    {attribute	'TcLinkTo'	:=	'.Status:=TIIB[K4S8_DRL_03_E18_EL6021]^COM TxPDO-Map Inputs^Status;
                                 .D[0]:=TIIB[K4S8_DRL_03_E18_EL6021]^COM TxPDO-Map Inputs^Data In 0;
                                 .D[1]:=TIIB[K4S8_DRL_03_E18_EL6021]^COM TxPDO-Map Inputs^Data In 1;
                                 .D[2]:=TIIB[K4S8_DRL_03_E18_EL6021]^COM TxPDO-Map Inputs^Data In 2;
                                 .D[3]:=TIIB[K4S8_DRL_03_E18_EL6021]^COM TxPDO-Map Inputs^Data In 3;
                                 .D[4]:=TIIB[K4S8_DRL_03_E18_EL6021]^COM TxPDO-Map Inputs^Data In 4;
                                 .D[5]:=TIIB[K4S8_DRL_03_E18_EL6021]^COM TxPDO-Map Inputs^Data In 5;
                                 .D[6]:=TIIB[K4S8_DRL_03_E18_EL6021]^COM TxPDO-Map Inputs^Data In 6;
                                 .D[7]:=TIIB[K4S8_DRL_03_E18_EL6021]^COM TxPDO-Map Inputs^Data In 7;
                                 .D[8]:=TIIB[K4S8_DRL_03_E18_EL6021]^COM TxPDO-Map Inputs^Data In 8;
                                 .D[9]:=TIIB[K4S8_DRL_03_E18_EL6021]^COM TxPDO-Map Inputs^Data In 9;
                                 .D[10]:=TIIB[K4S8_DRL_03_E18_EL6021]^COM TxPDO-Map Inputs^Data In 10;
                                 .D[11]:=TIIB[K4S8_DRL_03_E18_EL6021]^COM TxPDO-Map Inputs^Data In 11;
                                 .D[12]:=TIIB[K4S8_DRL_03_E18_EL6021]^COM TxPDO-Map Inputs^Data In 12;
                                 .D[13]:=TIIB[K4S8_DRL_03_E18_EL6021]^COM TxPDO-Map Inputs^Data In 13;
                                 .D[14]:=TIIB[K4S8_DRL_03_E18_EL6021]^COM TxPDO-Map Inputs^Data In 14;
                                 .D[15]:=TIIB[K4S8_DRL_03_E18_EL6021]^COM TxPDO-Map Inputs^Data In 15;
                                 .D[16]:=TIIB[K4S8_DRL_03_E18_EL6021]^COM TxPDO-Map Inputs^Data In 16;
                                 .D[17]:=TIIB[K4S8_DRL_03_E18_EL6021]^COM TxPDO-Map Inputs^Data In 17;
                                 .D[18]:=TIIB[K4S8_DRL_03_E18_EL6021]^COM TxPDO-Map Inputs^Data In 18;
                                 .D[19]:=TIIB[K4S8_DRL_03_E18_EL6021]^COM TxPDO-Map Inputs^Data In 19;
                                 .D[20]:=TIIB[K4S8_DRL_03_E18_EL6021]^COM TxPDO-Map Inputs^Data In 20;
                                 .D[21]:=TIIB[K4S8_DRL_03_E18_EL6021]^COM TxPDO-Map Inputs^Data In 21
    '}
    stComIn_DREAM_DP1_PTM_01 AT %I* : EL6inData22B;

    {attribute 'TcLinkTo'	:=	'.Ctrl:=TIIB[K4S8_DRL_03_E18_EL6021]^COM RxPDO-Map Outputs^Ctrl;
                                 .D[0]:=TIIB[K4S8_DRL_03_E18_EL6021]^COM RxPDO-Map Outputs^Data Out 0;
                                 .D[1]:=TIIB[K4S8_DRL_03_E18_EL6021]^COM RxPDO-Map Outputs^Data Out 1;
                                 .D[2]:=TIIB[K4S8_DRL_03_E18_EL6021]^COM RxPDO-Map Outputs^Data Out 2;
                                 .D[3]:=TIIB[K4S8_DRL_03_E18_EL6021]^COM RxPDO-Map Outputs^Data Out 3;
                                 .D[4]:=TIIB[K4S8_DRL_03_E18_EL6021]^COM RxPDO-Map Outputs^Data Out 4;
                                 .D[5]:=TIIB[K4S8_DRL_03_E18_EL6021]^COM RxPDO-Map Outputs^Data Out 5;
                                 .D[6]:=TIIB[K4S8_DRL_03_E18_EL6021]^COM RxPDO-Map Outputs^Data Out 6;
                                 .D[7]:=TIIB[K4S8_DRL_03_E18_EL6021]^COM RxPDO-Map Outputs^Data Out 7;
                                 .D[8]:=TIIB[K4S8_DRL_03_E18_EL6021]^COM RxPDO-Map Outputs^Data Out 8;
                                 .D[9]:=TIIB[K4S8_DRL_03_E18_EL6021]^COM RxPDO-Map Outputs^Data Out 9;
                                 .D[10]:=TIIB[K4S8_DRL_03_E18_EL6021]^COM RxPDO-Map Outputs^Data Out 10;
                                 .D[11]:=TIIB[K4S8_DRL_03_E18_EL6021]^COM RxPDO-Map Outputs^Data Out 11;
                                 .D[12]:=TIIB[K4S8_DRL_03_E18_EL6021]^COM RxPDO-Map Outputs^Data Out 12;
                                 .D[13]:=TIIB[K4S8_DRL_03_E18_EL6021]^COM RxPDO-Map Outputs^Data Out 13;
                                 .D[14]:=TIIB[K4S8_DRL_03_E18_EL6021]^COM RxPDO-Map Outputs^Data Out 14;
                                 .D[15]:=TIIB[K4S8_DRL_03_E18_EL6021]^COM RxPDO-Map Outputs^Data Out 15;
                                 .D[16]:=TIIB[K4S8_DRL_03_E18_EL6021]^COM RxPDO-Map Outputs^Data Out 16;
                                 .D[17]:=TIIB[K4S8_DRL_03_E18_EL6021]^COM RxPDO-Map Outputs^Data Out 17;
                                 .D[18]:=TIIB[K4S8_DRL_03_E18_EL6021]^COM RxPDO-Map Outputs^Data Out 18;
                                 .D[19]:=TIIB[K4S8_DRL_03_E18_EL6021]^COM RxPDO-Map Outputs^Data Out 19;
                                 .D[20]:=TIIB[K4S8_DRL_03_E18_EL6021]^COM RxPDO-Map Outputs^Data Out 20;
                                 .D[21]:=TIIB[K4S8_DRL_03_E18_EL6021]^COM RxPDO-Map Outputs^Data Out 21
    '}
    stComOut_DREAM_DP1_PTM_01 AT %Q* : EL6outData22B;

    {attribute	'TcLinkTo'	:=	'.Status:=TIIB[R20_DRL_03_E9_EL6001]^COM Inputs^Status;
                                 .D[0]:=TIIB[R20_DRL_03_E9_EL6001]^COM Inputs^Data In 0;
                                 .D[1]:=TIIB[R20_DRL_03_E9_EL6001]^COM Inputs^Data In 1;
                                 .D[2]:=TIIB[R20_DRL_03_E9_EL6001]^COM Inputs^Data In 2;
                                 .D[3]:=TIIB[R20_DRL_03_E9_EL6001]^COM Inputs^Data In 3;
                                 .D[4]:=TIIB[R20_DRL_03_E9_EL6001]^COM Inputs^Data In 4;
                                 .D[5]:=TIIB[R20_DRL_03_E9_EL6001]^COM Inputs^Data In 5;
                                 .D[6]:=TIIB[R20_DRL_03_E9_EL6001]^COM Inputs^Data In 6;
                                 .D[7]:=TIIB[R20_DRL_03_E9_EL6001]^COM Inputs^Data In 7;
                                 .D[8]:=TIIB[R20_DRL_03_E9_EL6001]^COM Inputs^Data In 8;
                                 .D[9]:=TIIB[R20_DRL_03_E9_EL6001]^COM Inputs^Data In 9;
                                 .D[10]:=TIIB[R20_DRL_03_E9_EL6001]^COM Inputs^Data In 10;
                                 .D[11]:=TIIB[R20_DRL_03_E9_EL6001]^COM Inputs^Data In 11;
                                 .D[12]:=TIIB[R20_DRL_03_E9_EL6001]^COM Inputs^Data In 12;
                                 .D[13]:=TIIB[R20_DRL_03_E9_EL6001]^COM Inputs^Data In 13;
                                 .D[14]:=TIIB[R20_DRL_03_E9_EL6001]^COM Inputs^Data In 14;
                                 .D[15]:=TIIB[R20_DRL_03_E9_EL6001]^COM Inputs^Data In 15;
                                 .D[16]:=TIIB[R20_DRL_03_E9_EL6001]^COM Inputs^Data In 16;
                                 .D[17]:=TIIB[R20_DRL_03_E9_EL6001]^COM Inputs^Data In 17;
                                 .D[18]:=TIIB[R20_DRL_03_E9_EL6001]^COM Inputs^Data In 18;
                                 .D[19]:=TIIB[R20_DRL_03_E9_EL6001]^COM Inputs^Data In 19;
                                 .D[20]:=TIIB[R20_DRL_03_E9_EL6001]^COM Inputs^Data In 20;
                                 .D[21]:=TIIB[R20_DRL_03_E9_EL6001]^COM Inputs^Data In 21
    '}
    stComIn_DREAM_DP2_PTM_01 AT %I* : EL6inData22B;

    {attribute 'TcLinkTo'	:=	'.Ctrl:=TIIB[R20_DRL_03_E9_EL6001]^COM Outputs^Ctrl;
                                 .D[0]:=TIIB[R20_DRL_03_E9_EL6001]^COM Outputs^Data Out 0;
                                 .D[1]:=TIIB[R20_DRL_03_E9_EL6001]^COM Outputs^Data Out 1;
                                 .D[2]:=TIIB[R20_DRL_03_E9_EL6001]^COM Outputs^Data Out 2;
                                 .D[3]:=TIIB[R20_DRL_03_E9_EL6001]^COM Outputs^Data Out 3;
                                 .D[4]:=TIIB[R20_DRL_03_E9_EL6001]^COM Outputs^Data Out 4;
                                 .D[5]:=TIIB[R20_DRL_03_E9_EL6001]^COM Outputs^Data Out 5;
                                 .D[6]:=TIIB[R20_DRL_03_E9_EL6001]^COM Outputs^Data Out 6;
                                 .D[7]:=TIIB[R20_DRL_03_E9_EL6001]^COM Outputs^Data Out 7;
                                 .D[8]:=TIIB[R20_DRL_03_E9_EL6001]^COM Outputs^Data Out 8;
                                 .D[9]:=TIIB[R20_DRL_03_E9_EL6001]^COM Outputs^Data Out 9;
                                 .D[10]:=TIIB[R20_DRL_03_E9_EL6001]^COM Outputs^Data Out 10;
                                 .D[11]:=TIIB[R20_DRL_03_E9_EL6001]^COM Outputs^Data Out 11;
                                 .D[12]:=TIIB[R20_DRL_03_E9_EL6001]^COM Outputs^Data Out 12;
                                 .D[13]:=TIIB[R20_DRL_03_E9_EL6001]^COM Outputs^Data Out 13;
                                 .D[14]:=TIIB[R20_DRL_03_E9_EL6001]^COM Outputs^Data Out 14;
                                 .D[15]:=TIIB[R20_DRL_03_E9_EL6001]^COM Outputs^Data Out 15;
                                 .D[16]:=TIIB[R20_DRL_03_E9_EL6001]^COM Outputs^Data Out 16;
                                 .D[17]:=TIIB[R20_DRL_03_E9_EL6001]^COM Outputs^Data Out 17;
                                 .D[18]:=TIIB[R20_DRL_03_E9_EL6001]^COM Outputs^Data Out 18;
                                 .D[19]:=TIIB[R20_DRL_03_E9_EL6001]^COM Outputs^Data Out 19;
                                 .D[20]:=TIIB[R20_DRL_03_E9_EL6001]^COM Outputs^Data Out 20;
                                 .D[21]:=TIIB[R20_DRL_03_E9_EL6001]^COM Outputs^Data Out 21
    '}
    stComOut_DREAM_DP2_PTM_01 AT %Q* : EL6outData22B;

    {attribute	'TcLinkTo'	:=	'.Status:=TIIB[R20_DRL_03_E10_EL6001]^COM Inputs^Status;
                                 .D[0]:=TIIB[R20_DRL_03_E10_EL6001]^COM Inputs^Data In 0;
                                 .D[1]:=TIIB[R20_DRL_03_E10_EL6001]^COM Inputs^Data In 1;
                                 .D[2]:=TIIB[R20_DRL_03_E10_EL6001]^COM Inputs^Data In 2;
                                 .D[3]:=TIIB[R20_DRL_03_E10_EL6001]^COM Inputs^Data In 3;
                                 .D[4]:=TIIB[R20_DRL_03_E10_EL6001]^COM Inputs^Data In 4;
                                 .D[5]:=TIIB[R20_DRL_03_E10_EL6001]^COM Inputs^Data In 5;
                                 .D[6]:=TIIB[R20_DRL_03_E10_EL6001]^COM Inputs^Data In 6;
                                 .D[7]:=TIIB[R20_DRL_03_E10_EL6001]^COM Inputs^Data In 7;
                                 .D[8]:=TIIB[R20_DRL_03_E10_EL6001]^COM Inputs^Data In 8;
                                 .D[9]:=TIIB[R20_DRL_03_E10_EL6001]^COM Inputs^Data In 9;
                                 .D[10]:=TIIB[R20_DRL_03_E10_EL6001]^COM Inputs^Data In 10;
                                 .D[11]:=TIIB[R20_DRL_03_E10_EL6001]^COM Inputs^Data In 11;
                                 .D[12]:=TIIB[R20_DRL_03_E10_EL6001]^COM Inputs^Data In 12;
                                 .D[13]:=TIIB[R20_DRL_03_E10_EL6001]^COM Inputs^Data In 13;
                                 .D[14]:=TIIB[R20_DRL_03_E10_EL6001]^COM Inputs^Data In 14;
                                 .D[15]:=TIIB[R20_DRL_03_E10_EL6001]^COM Inputs^Data In 15;
                                 .D[16]:=TIIB[R20_DRL_03_E10_EL6001]^COM Inputs^Data In 16;
                                 .D[17]:=TIIB[R20_DRL_03_E10_EL6001]^COM Inputs^Data In 17;
                                 .D[18]:=TIIB[R20_DRL_03_E10_EL6001]^COM Inputs^Data In 18;
                                 .D[19]:=TIIB[R20_DRL_03_E10_EL6001]^COM Inputs^Data In 19;
                                 .D[20]:=TIIB[R20_DRL_03_E10_EL6001]^COM Inputs^Data In 20;
                                 .D[21]:=TIIB[R20_DRL_03_E10_EL6001]^COM Inputs^Data In 21
    '}
    stComIn_DREAM_DP3_PTM_01 AT %I* : EL6inData22B;

    {attribute 'TcLinkTo'	:=	'.Ctrl:=TIIB[R20_DRL_03_E10_EL6001]^COM Outputs^Ctrl;
                                 .D[0]:=TIIB[R20_DRL_03_E10_EL6001]^COM Outputs^Data Out 0;
                                 .D[1]:=TIIB[R20_DRL_03_E10_EL6001]^COM Outputs^Data Out 1;
                                 .D[2]:=TIIB[R20_DRL_03_E10_EL6001]^COM Outputs^Data Out 2;
                                 .D[3]:=TIIB[R20_DRL_03_E10_EL6001]^COM Outputs^Data Out 3;
                                 .D[4]:=TIIB[R20_DRL_03_E10_EL6001]^COM Outputs^Data Out 4;
                                 .D[5]:=TIIB[R20_DRL_03_E10_EL6001]^COM Outputs^Data Out 5;
                                 .D[6]:=TIIB[R20_DRL_03_E10_EL6001]^COM Outputs^Data Out 6;
                                 .D[7]:=TIIB[R20_DRL_03_E10_EL6001]^COM Outputs^Data Out 7;
                                 .D[8]:=TIIB[R20_DRL_03_E10_EL6001]^COM Outputs^Data Out 8;
                                 .D[9]:=TIIB[R20_DRL_03_E10_EL6001]^COM Outputs^Data Out 9;
                                 .D[10]:=TIIB[R20_DRL_03_E10_EL6001]^COM Outputs^Data Out 10;
                                 .D[11]:=TIIB[R20_DRL_03_E10_EL6001]^COM Outputs^Data Out 11;
                                 .D[12]:=TIIB[R20_DRL_03_E10_EL6001]^COM Outputs^Data Out 12;
                                 .D[13]:=TIIB[R20_DRL_03_E10_EL6001]^COM Outputs^Data Out 13;
                                 .D[14]:=TIIB[R20_DRL_03_E10_EL6001]^COM Outputs^Data Out 14;
                                 .D[15]:=TIIB[R20_DRL_03_E10_EL6001]^COM Outputs^Data Out 15;
                                 .D[16]:=TIIB[R20_DRL_03_E10_EL6001]^COM Outputs^Data Out 16;
                                 .D[17]:=TIIB[R20_DRL_03_E10_EL6001]^COM Outputs^Data Out 17;
                                 .D[18]:=TIIB[R20_DRL_03_E10_EL6001]^COM Outputs^Data Out 18;
                                 .D[19]:=TIIB[R20_DRL_03_E10_EL6001]^COM Outputs^Data Out 19;
                                 .D[20]:=TIIB[R20_DRL_03_E10_EL6001]^COM Outputs^Data Out 20;
                                 .D[21]:=TIIB[R20_DRL_03_E10_EL6001]^COM Outputs^Data Out 21
    '}
    stComOut_DREAM_DP3_PTM_01 AT %Q* : EL6outData22B;

    {attribute	'TcLinkTo'	:=	'.Status:=TIIB[R20_DRL_03_E11_EL6001]^COM Inputs^Status;
                                 .D[0]:=TIIB[R20_DRL_03_E11_EL6001]^COM Inputs^Data In 0;
                                 .D[1]:=TIIB[R20_DRL_03_E11_EL6001]^COM Inputs^Data In 1;
                                 .D[2]:=TIIB[R20_DRL_03_E11_EL6001]^COM Inputs^Data In 2;
                                 .D[3]:=TIIB[R20_DRL_03_E11_EL6001]^COM Inputs^Data In 3;
                                 .D[4]:=TIIB[R20_DRL_03_E11_EL6001]^COM Inputs^Data In 4;
                                 .D[5]:=TIIB[R20_DRL_03_E11_EL6001]^COM Inputs^Data In 5;
                                 .D[6]:=TIIB[R20_DRL_03_E11_EL6001]^COM Inputs^Data In 6;
                                 .D[7]:=TIIB[R20_DRL_03_E11_EL6001]^COM Inputs^Data In 7;
                                 .D[8]:=TIIB[R20_DRL_03_E11_EL6001]^COM Inputs^Data In 8;
                                 .D[9]:=TIIB[R20_DRL_03_E11_EL6001]^COM Inputs^Data In 9;
                                 .D[10]:=TIIB[R20_DRL_03_E11_EL6001]^COM Inputs^Data In 10;
                                 .D[11]:=TIIB[R20_DRL_03_E11_EL6001]^COM Inputs^Data In 11;
                                 .D[12]:=TIIB[R20_DRL_03_E11_EL6001]^COM Inputs^Data In 12;
                                 .D[13]:=TIIB[R20_DRL_03_E11_EL6001]^COM Inputs^Data In 13;
                                 .D[14]:=TIIB[R20_DRL_03_E11_EL6001]^COM Inputs^Data In 14;
                                 .D[15]:=TIIB[R20_DRL_03_E11_EL6001]^COM Inputs^Data In 15;
                                 .D[16]:=TIIB[R20_DRL_03_E11_EL6001]^COM Inputs^Data In 16;
                                 .D[17]:=TIIB[R20_DRL_03_E11_EL6001]^COM Inputs^Data In 17;
                                 .D[18]:=TIIB[R20_DRL_03_E11_EL6001]^COM Inputs^Data In 18;
                                 .D[19]:=TIIB[R20_DRL_03_E11_EL6001]^COM Inputs^Data In 19;
                                 .D[20]:=TIIB[R20_DRL_03_E11_EL6001]^COM Inputs^Data In 20;
                                 .D[21]:=TIIB[R20_DRL_03_E11_EL6001]^COM Inputs^Data In 21
    '}
    stComIn_DREAM_MC_PTM_01 AT %I* : EL6inData22B;

    {attribute 'TcLinkTo'	:=	'.Ctrl:=TIIB[R20_DRL_03_E11_EL6001]^COM Outputs^Ctrl;
                                 .D[0]:=TIIB[R20_DRL_03_E11_EL6001]^COM Outputs^Data Out 0;
                                 .D[1]:=TIIB[R20_DRL_03_E11_EL6001]^COM Outputs^Data Out 1;
                                 .D[2]:=TIIB[R20_DRL_03_E11_EL6001]^COM Outputs^Data Out 2;
                                 .D[3]:=TIIB[R20_DRL_03_E11_EL6001]^COM Outputs^Data Out 3;
                                 .D[4]:=TIIB[R20_DRL_03_E11_EL6001]^COM Outputs^Data Out 4;
                                 .D[5]:=TIIB[R20_DRL_03_E11_EL6001]^COM Outputs^Data Out 5;
                                 .D[6]:=TIIB[R20_DRL_03_E11_EL6001]^COM Outputs^Data Out 6;
                                 .D[7]:=TIIB[R20_DRL_03_E11_EL6001]^COM Outputs^Data Out 7;
                                 .D[8]:=TIIB[R20_DRL_03_E11_EL6001]^COM Outputs^Data Out 8;
                                 .D[9]:=TIIB[R20_DRL_03_E11_EL6001]^COM Outputs^Data Out 9;
                                 .D[10]:=TIIB[R20_DRL_03_E11_EL6001]^COM Outputs^Data Out 10;
                                 .D[11]:=TIIB[R20_DRL_03_E11_EL6001]^COM Outputs^Data Out 11;
                                 .D[12]:=TIIB[R20_DRL_03_E11_EL6001]^COM Outputs^Data Out 12;
                                 .D[13]:=TIIB[R20_DRL_03_E11_EL6001]^COM Outputs^Data Out 13;
                                 .D[14]:=TIIB[R20_DRL_03_E11_EL6001]^COM Outputs^Data Out 14;
                                 .D[15]:=TIIB[R20_DRL_03_E11_EL6001]^COM Outputs^Data Out 15;
                                 .D[16]:=TIIB[R20_DRL_03_E11_EL6001]^COM Outputs^Data Out 16;
                                 .D[17]:=TIIB[R20_DRL_03_E11_EL6001]^COM Outputs^Data Out 17;
                                 .D[18]:=TIIB[R20_DRL_03_E11_EL6001]^COM Outputs^Data Out 18;
                                 .D[19]:=TIIB[R20_DRL_03_E11_EL6001]^COM Outputs^Data Out 19;
                                 .D[20]:=TIIB[R20_DRL_03_E11_EL6001]^COM Outputs^Data Out 20;
                                 .D[21]:=TIIB[R20_DRL_03_E11_EL6001]^COM Outputs^Data Out 21
    '}
    stComOut_DREAM_MC_PTM_01 AT %Q* : EL6outData22B;

    {attribute	'TcLinkTo'	:=	'.Status:=TIIB[R20_DRL_03_E12_EL6001]^COM Inputs^Status;
                                 .D[0]:=TIIB[R20_DRL_03_E12_EL6001]^COM Inputs^Data In 0;
                                 .D[1]:=TIIB[R20_DRL_03_E12_EL6001]^COM Inputs^Data In 1;
                                 .D[2]:=TIIB[R20_DRL_03_E12_EL6001]^COM Inputs^Data In 2;
                                 .D[3]:=TIIB[R20_DRL_03_E12_EL6001]^COM Inputs^Data In 3;
                                 .D[4]:=TIIB[R20_DRL_03_E12_EL6001]^COM Inputs^Data In 4;
                                 .D[5]:=TIIB[R20_DRL_03_E12_EL6001]^COM Inputs^Data In 5;
                                 .D[6]:=TIIB[R20_DRL_03_E12_EL6001]^COM Inputs^Data In 6;
                                 .D[7]:=TIIB[R20_DRL_03_E12_EL6001]^COM Inputs^Data In 7;
                                 .D[8]:=TIIB[R20_DRL_03_E12_EL6001]^COM Inputs^Data In 8;
                                 .D[9]:=TIIB[R20_DRL_03_E12_EL6001]^COM Inputs^Data In 9;
                                 .D[10]:=TIIB[R20_DRL_03_E12_EL6001]^COM Inputs^Data In 10;
                                 .D[11]:=TIIB[R20_DRL_03_E12_EL6001]^COM Inputs^Data In 11;
                                 .D[12]:=TIIB[R20_DRL_03_E12_EL6001]^COM Inputs^Data In 12;
                                 .D[13]:=TIIB[R20_DRL_03_E12_EL6001]^COM Inputs^Data In 13;
                                 .D[14]:=TIIB[R20_DRL_03_E12_EL6001]^COM Inputs^Data In 14;
                                 .D[15]:=TIIB[R20_DRL_03_E12_EL6001]^COM Inputs^Data In 15;
                                 .D[16]:=TIIB[R20_DRL_03_E12_EL6001]^COM Inputs^Data In 16;
                                 .D[17]:=TIIB[R20_DRL_03_E12_EL6001]^COM Inputs^Data In 17;
                                 .D[18]:=TIIB[R20_DRL_03_E12_EL6001]^COM Inputs^Data In 18;
                                 .D[19]:=TIIB[R20_DRL_03_E12_EL6001]^COM Inputs^Data In 19;
                                 .D[20]:=TIIB[R20_DRL_03_E12_EL6001]^COM Inputs^Data In 20;
                                 .D[21]:=TIIB[R20_DRL_03_E12_EL6001]^COM Inputs^Data In 21
    '}
    stComIn_DREAM_MC_PTM_02 AT %I* : EL6inData22B;

    {attribute 'TcLinkTo'	:=	'.Ctrl:=TIIB[R20_DRL_03_E12_EL6001]^COM Outputs^Ctrl;
                                 .D[0]:=TIIB[R20_DRL_03_E12_EL6001]^COM Outputs^Data Out 0;
                                 .D[1]:=TIIB[R20_DRL_03_E12_EL6001]^COM Outputs^Data Out 1;
                                 .D[2]:=TIIB[R20_DRL_03_E12_EL6001]^COM Outputs^Data Out 2;
                                 .D[3]:=TIIB[R20_DRL_03_E12_EL6001]^COM Outputs^Data Out 3;
                                 .D[4]:=TIIB[R20_DRL_03_E12_EL6001]^COM Outputs^Data Out 4;
                                 .D[5]:=TIIB[R20_DRL_03_E12_EL6001]^COM Outputs^Data Out 5;
                                 .D[6]:=TIIB[R20_DRL_03_E12_EL6001]^COM Outputs^Data Out 6;
                                 .D[7]:=TIIB[R20_DRL_03_E12_EL6001]^COM Outputs^Data Out 7;
                                 .D[8]:=TIIB[R20_DRL_03_E12_EL6001]^COM Outputs^Data Out 8;
                                 .D[9]:=TIIB[R20_DRL_03_E12_EL6001]^COM Outputs^Data Out 9;
                                 .D[10]:=TIIB[R20_DRL_03_E12_EL6001]^COM Outputs^Data Out 10;
                                 .D[11]:=TIIB[R20_DRL_03_E12_EL6001]^COM Outputs^Data Out 11;
                                 .D[12]:=TIIB[R20_DRL_03_E12_EL6001]^COM Outputs^Data Out 12;
                                 .D[13]:=TIIB[R20_DRL_03_E12_EL6001]^COM Outputs^Data Out 13;
                                 .D[14]:=TIIB[R20_DRL_03_E12_EL6001]^COM Outputs^Data Out 14;
                                 .D[15]:=TIIB[R20_DRL_03_E12_EL6001]^COM Outputs^Data Out 15;
                                 .D[16]:=TIIB[R20_DRL_03_E12_EL6001]^COM Outputs^Data Out 16;
                                 .D[17]:=TIIB[R20_DRL_03_E12_EL6001]^COM Outputs^Data Out 17;
                                 .D[18]:=TIIB[R20_DRL_03_E12_EL6001]^COM Outputs^Data Out 18;
                                 .D[19]:=TIIB[R20_DRL_03_E12_EL6001]^COM Outputs^Data Out 19;
                                 .D[20]:=TIIB[R20_DRL_03_E12_EL6001]^COM Outputs^Data Out 20;
                                 .D[21]:=TIIB[R20_DRL_03_E12_EL6001]^COM Outputs^Data Out 21
    '}
    stComOut_DREAM_MC_PTM_02 AT %Q* : EL6outData22B;

    {attribute	'TcLinkTo'	:=	'.Status:=TIIB[K4S8_DRL_04_E7_EL6001]^COM Inputs^Status;
                                 .D[0]:=TIIB[K4S8_DRL_04_E7_EL6001]^COM Inputs^Data In 0;
                                 .D[1]:=TIIB[K4S8_DRL_04_E7_EL6001]^COM Inputs^Data In 1;
                                 .D[2]:=TIIB[K4S8_DRL_04_E7_EL6001]^COM Inputs^Data In 2;
                                 .D[3]:=TIIB[K4S8_DRL_04_E7_EL6001]^COM Inputs^Data In 3;
                                 .D[4]:=TIIB[K4S8_DRL_04_E7_EL6001]^COM Inputs^Data In 4;
                                 .D[5]:=TIIB[K4S8_DRL_04_E7_EL6001]^COM Inputs^Data In 5;
                                 .D[6]:=TIIB[K4S8_DRL_04_E7_EL6001]^COM Inputs^Data In 6;
                                 .D[7]:=TIIB[K4S8_DRL_04_E7_EL6001]^COM Inputs^Data In 7;
                                 .D[8]:=TIIB[K4S8_DRL_04_E7_EL6001]^COM Inputs^Data In 8;
                                 .D[9]:=TIIB[K4S8_DRL_04_E7_EL6001]^COM Inputs^Data In 9;
                                 .D[10]:=TIIB[K4S8_DRL_04_E7_EL6001]^COM Inputs^Data In 10;
                                 .D[11]:=TIIB[K4S8_DRL_04_E7_EL6001]^COM Inputs^Data In 11;
                                 .D[12]:=TIIB[K4S8_DRL_04_E7_EL6001]^COM Inputs^Data In 12;
                                 .D[13]:=TIIB[K4S8_DRL_04_E7_EL6001]^COM Inputs^Data In 13;
                                 .D[14]:=TIIB[K4S8_DRL_04_E7_EL6001]^COM Inputs^Data In 14;
                                 .D[15]:=TIIB[K4S8_DRL_04_E7_EL6001]^COM Inputs^Data In 15;
                                 .D[16]:=TIIB[K4S8_DRL_04_E7_EL6001]^COM Inputs^Data In 16;
                                 .D[17]:=TIIB[K4S8_DRL_04_E7_EL6001]^COM Inputs^Data In 17;
                                 .D[18]:=TIIB[K4S8_DRL_04_E7_EL6001]^COM Inputs^Data In 18;
                                 .D[19]:=TIIB[K4S8_DRL_04_E7_EL6001]^COM Inputs^Data In 19;
                                 .D[20]:=TIIB[K4S8_DRL_04_E7_EL6001]^COM Inputs^Data In 20;
                                 .D[21]:=TIIB[K4S8_DRL_04_E7_EL6001]^COM Inputs^Data In 21
    '}
    stComIn_DREAM_CAT1_PTM_01 AT %I* : EL6inData22B;

    {attribute 'TcLinkTo'	:=	'.Ctrl:=TIIB[K4S8_DRL_04_E7_EL6001]^COM Outputs^Ctrl;
                                 .D[0]:=TIIB[K4S8_DRL_04_E7_EL6001]^COM Outputs^Data Out 0;
                                 .D[1]:=TIIB[K4S8_DRL_04_E7_EL6001]^COM Outputs^Data Out 1;
                                 .D[2]:=TIIB[K4S8_DRL_04_E7_EL6001]^COM Outputs^Data Out 2;
                                 .D[3]:=TIIB[K4S8_DRL_04_E7_EL6001]^COM Outputs^Data Out 3;
                                 .D[4]:=TIIB[K4S8_DRL_04_E7_EL6001]^COM Outputs^Data Out 4;
                                 .D[5]:=TIIB[K4S8_DRL_04_E7_EL6001]^COM Outputs^Data Out 5;
                                 .D[6]:=TIIB[K4S8_DRL_04_E7_EL6001]^COM Outputs^Data Out 6;
                                 .D[7]:=TIIB[K4S8_DRL_04_E7_EL6001]^COM Outputs^Data Out 7;
                                 .D[8]:=TIIB[K4S8_DRL_04_E7_EL6001]^COM Outputs^Data Out 8;
                                 .D[9]:=TIIB[K4S8_DRL_04_E7_EL6001]^COM Outputs^Data Out 9;
                                 .D[10]:=TIIB[K4S8_DRL_04_E7_EL6001]^COM Outputs^Data Out 10;
                                 .D[11]:=TIIB[K4S8_DRL_04_E7_EL6001]^COM Outputs^Data Out 11;
                                 .D[12]:=TIIB[K4S8_DRL_04_E7_EL6001]^COM Outputs^Data Out 12;
                                 .D[13]:=TIIB[K4S8_DRL_04_E7_EL6001]^COM Outputs^Data Out 13;
                                 .D[14]:=TIIB[K4S8_DRL_04_E7_EL6001]^COM Outputs^Data Out 14;
                                 .D[15]:=TIIB[K4S8_DRL_04_E7_EL6001]^COM Outputs^Data Out 15;
                                 .D[16]:=TIIB[K4S8_DRL_04_E7_EL6001]^COM Outputs^Data Out 16;
                                 .D[17]:=TIIB[K4S8_DRL_04_E7_EL6001]^COM Outputs^Data Out 17;
                                 .D[18]:=TIIB[K4S8_DRL_04_E7_EL6001]^COM Outputs^Data Out 18;
                                 .D[19]:=TIIB[K4S8_DRL_04_E7_EL6001]^COM Outputs^Data Out 19;
                                 .D[20]:=TIIB[K4S8_DRL_04_E7_EL6001]^COM Outputs^Data Out 20;
                                 .D[21]:=TIIB[K4S8_DRL_04_E7_EL6001]^COM Outputs^Data Out 21
    '}
    stComOut_DREAM_CAT1_PTM_01 AT %Q* : EL6outData22B;

    {attribute	'TcLinkTo'	:=	'.Status:=TIIB[K4S8_DRL_04_E8_EL6001]^COM Inputs^Status;
                                 .D[0]:=TIIB[K4S8_DRL_04_E8_EL6001]^COM Inputs^Data In 0;
                                 .D[1]:=TIIB[K4S8_DRL_04_E8_EL6001]^COM Inputs^Data In 1;
                                 .D[2]:=TIIB[K4S8_DRL_04_E8_EL6001]^COM Inputs^Data In 2;
                                 .D[3]:=TIIB[K4S8_DRL_04_E8_EL6001]^COM Inputs^Data In 3;
                                 .D[4]:=TIIB[K4S8_DRL_04_E8_EL6001]^COM Inputs^Data In 4;
                                 .D[5]:=TIIB[K4S8_DRL_04_E8_EL6001]^COM Inputs^Data In 5;
                                 .D[6]:=TIIB[K4S8_DRL_04_E8_EL6001]^COM Inputs^Data In 6;
                                 .D[7]:=TIIB[K4S8_DRL_04_E8_EL6001]^COM Inputs^Data In 7;
                                 .D[8]:=TIIB[K4S8_DRL_04_E8_EL6001]^COM Inputs^Data In 8;
                                 .D[9]:=TIIB[K4S8_DRL_04_E8_EL6001]^COM Inputs^Data In 9;
                                 .D[10]:=TIIB[K4S8_DRL_04_E8_EL6001]^COM Inputs^Data In 10;
                                 .D[11]:=TIIB[K4S8_DRL_04_E8_EL6001]^COM Inputs^Data In 11;
                                 .D[12]:=TIIB[K4S8_DRL_04_E8_EL6001]^COM Inputs^Data In 12;
                                 .D[13]:=TIIB[K4S8_DRL_04_E8_EL6001]^COM Inputs^Data In 13;
                                 .D[14]:=TIIB[K4S8_DRL_04_E8_EL6001]^COM Inputs^Data In 14;
                                 .D[15]:=TIIB[K4S8_DRL_04_E8_EL6001]^COM Inputs^Data In 15;
                                 .D[16]:=TIIB[K4S8_DRL_04_E8_EL6001]^COM Inputs^Data In 16;
                                 .D[17]:=TIIB[K4S8_DRL_04_E8_EL6001]^COM Inputs^Data In 17;
                                 .D[18]:=TIIB[K4S8_DRL_04_E8_EL6001]^COM Inputs^Data In 18;
                                 .D[19]:=TIIB[K4S8_DRL_04_E8_EL6001]^COM Inputs^Data In 19;
                                 .D[20]:=TIIB[K4S8_DRL_04_E8_EL6001]^COM Inputs^Data In 20;
                                 .D[21]:=TIIB[K4S8_DRL_04_E8_EL6001]^COM Inputs^Data In 21
    '}
    stComIn_DREAM_CAT2_PTM_01 AT %I* : EL6inData22B;

    {attribute 'TcLinkTo'	:=	'.Ctrl:=TIIB[K4S8_DRL_04_E8_EL6001]^COM Outputs^Ctrl;
                                 .D[0]:=TIIB[K4S8_DRL_04_E8_EL6001]^COM Outputs^Data Out 0;
                                 .D[1]:=TIIB[K4S8_DRL_04_E8_EL6001]^COM Outputs^Data Out 1;
                                 .D[2]:=TIIB[K4S8_DRL_04_E8_EL6001]^COM Outputs^Data Out 2;
                                 .D[3]:=TIIB[K4S8_DRL_04_E8_EL6001]^COM Outputs^Data Out 3;
                                 .D[4]:=TIIB[K4S8_DRL_04_E8_EL6001]^COM Outputs^Data Out 4;
                                 .D[5]:=TIIB[K4S8_DRL_04_E8_EL6001]^COM Outputs^Data Out 5;
                                 .D[6]:=TIIB[K4S8_DRL_04_E8_EL6001]^COM Outputs^Data Out 6;
                                 .D[7]:=TIIB[K4S8_DRL_04_E8_EL6001]^COM Outputs^Data Out 7;
                                 .D[8]:=TIIB[K4S8_DRL_04_E8_EL6001]^COM Outputs^Data Out 8;
                                 .D[9]:=TIIB[K4S8_DRL_04_E8_EL6001]^COM Outputs^Data Out 9;
                                 .D[10]:=TIIB[K4S8_DRL_04_E8_EL6001]^COM Outputs^Data Out 10;
                                 .D[11]:=TIIB[K4S8_DRL_04_E8_EL6001]^COM Outputs^Data Out 11;
                                 .D[12]:=TIIB[K4S8_DRL_04_E8_EL6001]^COM Outputs^Data Out 12;
                                 .D[13]:=TIIB[K4S8_DRL_04_E8_EL6001]^COM Outputs^Data Out 13;
                                 .D[14]:=TIIB[K4S8_DRL_04_E8_EL6001]^COM Outputs^Data Out 14;
                                 .D[15]:=TIIB[K4S8_DRL_04_E8_EL6001]^COM Outputs^Data Out 15;
                                 .D[16]:=TIIB[K4S8_DRL_04_E8_EL6001]^COM Outputs^Data Out 16;
                                 .D[17]:=TIIB[K4S8_DRL_04_E8_EL6001]^COM Outputs^Data Out 17;
                                 .D[18]:=TIIB[K4S8_DRL_04_E8_EL6001]^COM Outputs^Data Out 18;
                                 .D[19]:=TIIB[K4S8_DRL_04_E8_EL6001]^COM Outputs^Data Out 19;
                                 .D[20]:=TIIB[K4S8_DRL_04_E8_EL6001]^COM Outputs^Data Out 20;
                                 .D[21]:=TIIB[K4S8_DRL_04_E8_EL6001]^COM Outputs^Data Out 21
    '}
    stComOut_DREAM_CAT2_PTM_01 AT %Q* : EL6outData22B;

    {attribute	'TcLinkTo'	:=	'.Status:=TIIB[K4S8_DRL_04_E6_EL6001]^COM Inputs^Status;
                                 .D[0]:=TIIB[K4S8_DRL_04_E6_EL6001]^COM Inputs^Data In 0;
                                 .D[1]:=TIIB[K4S8_DRL_04_E6_EL6001]^COM Inputs^Data In 1;
                                 .D[2]:=TIIB[K4S8_DRL_04_E6_EL6001]^COM Inputs^Data In 2;
                                 .D[3]:=TIIB[K4S8_DRL_04_E6_EL6001]^COM Inputs^Data In 3;
                                 .D[4]:=TIIB[K4S8_DRL_04_E6_EL6001]^COM Inputs^Data In 4;
                                 .D[5]:=TIIB[K4S8_DRL_04_E6_EL6001]^COM Inputs^Data In 5;
                                 .D[6]:=TIIB[K4S8_DRL_04_E6_EL6001]^COM Inputs^Data In 6;
                                 .D[7]:=TIIB[K4S8_DRL_04_E6_EL6001]^COM Inputs^Data In 7;
                                 .D[8]:=TIIB[K4S8_DRL_04_E6_EL6001]^COM Inputs^Data In 8;
                                 .D[9]:=TIIB[K4S8_DRL_04_E6_EL6001]^COM Inputs^Data In 9;
                                 .D[10]:=TIIB[K4S8_DRL_04_E6_EL6001]^COM Inputs^Data In 10;
                                 .D[11]:=TIIB[K4S8_DRL_04_E6_EL6001]^COM Inputs^Data In 11;
                                 .D[12]:=TIIB[K4S8_DRL_04_E6_EL6001]^COM Inputs^Data In 12;
                                 .D[13]:=TIIB[K4S8_DRL_04_E6_EL6001]^COM Inputs^Data In 13;
                                 .D[14]:=TIIB[K4S8_DRL_04_E6_EL6001]^COM Inputs^Data In 14;
                                 .D[15]:=TIIB[K4S8_DRL_04_E6_EL6001]^COM Inputs^Data In 15;
                                 .D[16]:=TIIB[K4S8_DRL_04_E6_EL6001]^COM Inputs^Data In 16;
                                 .D[17]:=TIIB[K4S8_DRL_04_E6_EL6001]^COM Inputs^Data In 17;
                                 .D[18]:=TIIB[K4S8_DRL_04_E6_EL6001]^COM Inputs^Data In 18;
                                 .D[19]:=TIIB[K4S8_DRL_04_E6_EL6001]^COM Inputs^Data In 19;
                                 .D[20]:=TIIB[K4S8_DRL_04_E6_EL6001]^COM Inputs^Data In 20;
                                 .D[21]:=TIIB[K4S8_DRL_04_E6_EL6001]^COM Inputs^Data In 21
    '}
    stComIn_DREAM_ROUGH2_PTM_01 AT %I* : EL6inData22B;

    {attribute 'TcLinkTo'	:=	'.Ctrl:=TIIB[K4S8_DRL_04_E6_EL6001]^COM Outputs^Ctrl;
                                 .D[0]:=TIIB[K4S8_DRL_04_E6_EL6001]^COM Outputs^Data Out 0;
                                 .D[1]:=TIIB[K4S8_DRL_04_E6_EL6001]^COM Outputs^Data Out 1;
                                 .D[2]:=TIIB[K4S8_DRL_04_E6_EL6001]^COM Outputs^Data Out 2;
                                 .D[3]:=TIIB[K4S8_DRL_04_E6_EL6001]^COM Outputs^Data Out 3;
                                 .D[4]:=TIIB[K4S8_DRL_04_E6_EL6001]^COM Outputs^Data Out 4;
                                 .D[5]:=TIIB[K4S8_DRL_04_E6_EL6001]^COM Outputs^Data Out 5;
                                 .D[6]:=TIIB[K4S8_DRL_04_E6_EL6001]^COM Outputs^Data Out 6;
                                 .D[7]:=TIIB[K4S8_DRL_04_E6_EL6001]^COM Outputs^Data Out 7;
                                 .D[8]:=TIIB[K4S8_DRL_04_E6_EL6001]^COM Outputs^Data Out 8;
                                 .D[9]:=TIIB[K4S8_DRL_04_E6_EL6001]^COM Outputs^Data Out 9;
                                 .D[10]:=TIIB[K4S8_DRL_04_E6_EL6001]^COM Outputs^Data Out 10;
                                 .D[11]:=TIIB[K4S8_DRL_04_E6_EL6001]^COM Outputs^Data Out 11;
                                 .D[12]:=TIIB[K4S8_DRL_04_E6_EL6001]^COM Outputs^Data Out 12;
                                 .D[13]:=TIIB[K4S8_DRL_04_E6_EL6001]^COM Outputs^Data Out 13;
                                 .D[14]:=TIIB[K4S8_DRL_04_E6_EL6001]^COM Outputs^Data Out 14;
                                 .D[15]:=TIIB[K4S8_DRL_04_E6_EL6001]^COM Outputs^Data Out 15;
                                 .D[16]:=TIIB[K4S8_DRL_04_E6_EL6001]^COM Outputs^Data Out 16;
                                 .D[17]:=TIIB[K4S8_DRL_04_E6_EL6001]^COM Outputs^Data Out 17;
                                 .D[18]:=TIIB[K4S8_DRL_04_E6_EL6001]^COM Outputs^Data Out 18;
                                 .D[19]:=TIIB[K4S8_DRL_04_E6_EL6001]^COM Outputs^Data Out 19;
                                 .D[20]:=TIIB[K4S8_DRL_04_E6_EL6001]^COM Outputs^Data Out 20;
                                 .D[21]:=TIIB[K4S8_DRL_04_E6_EL6001]^COM Outputs^Data Out 21
    '}
    stComOut_DREAM_ROUGH2_PTM_01 AT %Q* : EL6outData22B;

    {attribute	'TcLinkTo'	:=	'.Status:=TIIB[K4S8_DRL_04_E17_EL6001]^COM Inputs^Status;
                                 .D[0]:=TIIB[K4S8_DRL_04_E17_EL6001]^COM Inputs^Data In 0;
                                 .D[1]:=TIIB[K4S8_DRL_04_E17_EL6001]^COM Inputs^Data In 1;
                                 .D[2]:=TIIB[K4S8_DRL_04_E17_EL6001]^COM Inputs^Data In 2;
                                 .D[3]:=TIIB[K4S8_DRL_04_E17_EL6001]^COM Inputs^Data In 3;
                                 .D[4]:=TIIB[K4S8_DRL_04_E17_EL6001]^COM Inputs^Data In 4;
                                 .D[5]:=TIIB[K4S8_DRL_04_E17_EL6001]^COM Inputs^Data In 5;
                                 .D[6]:=TIIB[K4S8_DRL_04_E17_EL6001]^COM Inputs^Data In 6;
                                 .D[7]:=TIIB[K4S8_DRL_04_E17_EL6001]^COM Inputs^Data In 7;
                                 .D[8]:=TIIB[K4S8_DRL_04_E17_EL6001]^COM Inputs^Data In 8;
                                 .D[9]:=TIIB[K4S8_DRL_04_E17_EL6001]^COM Inputs^Data In 9;
                                 .D[10]:=TIIB[K4S8_DRL_04_E17_EL6001]^COM Inputs^Data In 10;
                                 .D[11]:=TIIB[K4S8_DRL_04_E17_EL6001]^COM Inputs^Data In 11;
                                 .D[12]:=TIIB[K4S8_DRL_04_E17_EL6001]^COM Inputs^Data In 12;
                                 .D[13]:=TIIB[K4S8_DRL_04_E17_EL6001]^COM Inputs^Data In 13;
                                 .D[14]:=TIIB[K4S8_DRL_04_E17_EL6001]^COM Inputs^Data In 14;
                                 .D[15]:=TIIB[K4S8_DRL_04_E17_EL6001]^COM Inputs^Data In 15;
                                 .D[16]:=TIIB[K4S8_DRL_04_E17_EL6001]^COM Inputs^Data In 16;
                                 .D[17]:=TIIB[K4S8_DRL_04_E17_EL6001]^COM Inputs^Data In 17;
                                 .D[18]:=TIIB[K4S8_DRL_04_E17_EL6001]^COM Inputs^Data In 18;
                                 .D[19]:=TIIB[K4S8_DRL_04_E17_EL6001]^COM Inputs^Data In 19;
                                 .D[20]:=TIIB[K4S8_DRL_04_E17_EL6001]^COM Inputs^Data In 20;
                                 .D[21]:=TIIB[K4S8_DRL_04_E17_EL6001]^COM Inputs^Data In 21
    '}
    stComIn_DREAM_ROUGH2_PTM_02 AT %I* : EL6inData22B;

    {attribute 'TcLinkTo'	:=	'.Ctrl:=TIIB[K4S8_DRL_04_E17_EL6001]^COM Outputs^Ctrl;
                                 .D[0]:=TIIB[K4S8_DRL_04_E17_EL6001]^COM Outputs^Data Out 0;
                                 .D[1]:=TIIB[K4S8_DRL_04_E17_EL6001]^COM Outputs^Data Out 1;
                                 .D[2]:=TIIB[K4S8_DRL_04_E17_EL6001]^COM Outputs^Data Out 2;
                                 .D[3]:=TIIB[K4S8_DRL_04_E17_EL6001]^COM Outputs^Data Out 3;
                                 .D[4]:=TIIB[K4S8_DRL_04_E17_EL6001]^COM Outputs^Data Out 4;
                                 .D[5]:=TIIB[K4S8_DRL_04_E17_EL6001]^COM Outputs^Data Out 5;
                                 .D[6]:=TIIB[K4S8_DRL_04_E17_EL6001]^COM Outputs^Data Out 6;
                                 .D[7]:=TIIB[K4S8_DRL_04_E17_EL6001]^COM Outputs^Data Out 7;
                                 .D[8]:=TIIB[K4S8_DRL_04_E17_EL6001]^COM Outputs^Data Out 8;
                                 .D[9]:=TIIB[K4S8_DRL_04_E17_EL6001]^COM Outputs^Data Out 9;
                                 .D[10]:=TIIB[K4S8_DRL_04_E17_EL6001]^COM Outputs^Data Out 10;
                                 .D[11]:=TIIB[K4S8_DRL_04_E17_EL6001]^COM Outputs^Data Out 11;
                                 .D[12]:=TIIB[K4S8_DRL_04_E17_EL6001]^COM Outputs^Data Out 12;
                                 .D[13]:=TIIB[K4S8_DRL_04_E17_EL6001]^COM Outputs^Data Out 13;
                                 .D[14]:=TIIB[K4S8_DRL_04_E17_EL6001]^COM Outputs^Data Out 14;
                                 .D[15]:=TIIB[K4S8_DRL_04_E17_EL6001]^COM Outputs^Data Out 15;
                                 .D[16]:=TIIB[K4S8_DRL_04_E17_EL6001]^COM Outputs^Data Out 16;
                                 .D[17]:=TIIB[K4S8_DRL_04_E17_EL6001]^COM Outputs^Data Out 17;
                                 .D[18]:=TIIB[K4S8_DRL_04_E17_EL6001]^COM Outputs^Data Out 18;
                                 .D[19]:=TIIB[K4S8_DRL_04_E17_EL6001]^COM Outputs^Data Out 19;
                                 .D[20]:=TIIB[K4S8_DRL_04_E17_EL6001]^COM Outputs^Data Out 20;
                                 .D[21]:=TIIB[K4S8_DRL_04_E17_EL6001]^COM Outputs^Data Out 21
    '}
    stComOut_DREAM_ROUGH2_PTM_02 AT %Q* : EL6outData22B;
END_VAR

// ---- GVLs/GVL_TC.TcGVL
VAR_GLOBAL
    {attribute 'TcLinkTo' := 	'.iRaw 			:=	TIIB[K4S8_DRL_03_E22_EL3314]^TC Inputs Channel 1^Value;
                                 .bError  		:=	TIIB[K4S8_DRL_03_E22_EL3314]^TC Inputs Channel 1^Error;
                                 .bUnderrange 	:=	TIIB[K4S8_DRL_03_E22_EL3314]^TC Inputs Channel 1^Underrange;
                                 .bOverrange  	:=	TIIB[K4S8_DRL_03_E22_EL3314]^TC Inputs Channel 1^Overrange
    '}
    {attribute 'pytmc' := ' pv: DREAM:STC:01'}
    TC_01 : FB_TempSensor;

    {attribute 'TcLinkTo' := 	'.iRaw 			:=	TIIB[K4S8_DRL_03_E22_EL3314]^TC Inputs Channel 2^Value;
                                 .bError  		:=	TIIB[K4S8_DRL_03_E22_EL3314]^TC Inputs Channel 2^Status^Error;
                                 .bUnderrange 	:=	TIIB[K4S8_DRL_03_E22_EL3314]^TC Inputs Channel 2^Status^Underrange;
                                 .bOverrange  	:=	TIIB[K4S8_DRL_03_E22_EL3314]^TC Inputs Channel 2^Status^Overrange
    '}
    {attribute 'pytmc' := ' pv: DREAM:STC:02'}
    TC_02 : FB_TempSensor;

    {attribute 'TcLinkTo' := 	'.iRaw 			:=	TIIB[K4S8_DRL_03_E22_EL3314]^TC Inputs Channel 3^Value;
                                 .bError  		:=	TIIB[K4S8_DRL_03_E22_EL3314]^TC Inputs Channel 3^Status^Error;
                                 .bUnderrange 	:=	TIIB[K4S8_DRL_03_E22_EL3314]^TC Inputs Channel 3^Status^Underrange;
                                 .bOverrange  	:=	TIIB[K4S8_DRL_03_E22_EL3314]^TC Inputs Channel 3^Status^Overrange
    '}
    {attribute 'pytmc' := ' pv: DREAM:STC:03'}
    TC_03 : FB_TempSensor;

    {attribute 'TcLinkTo' := 	'.iRaw 			:=	TIIB[K4S8_DRL_03_E22_EL3314]^TC Inputs Channel 4^Value;
                                 .bError  		:=	TIIB[K4S8_DRL_03_E22_EL3314]^TC Inputs Channel 4^Status^Error;
                                 .bUnderrange 	:=	TIIB[K4S8_DRL_03_E22_EL3314]^TC Inputs Channel 4^Status^Underrange;
                                 .bOverrange  	:=	TIIB[K4S8_DRL_03_E22_EL3314]^TC Inputs Channel 4^Status^Overrange
    '}
    {attribute 'pytmc' := ' pv: DREAM:STC:04'}
    TC_04 : FB_TempSensor;

    {attribute 'TcLinkTo' := 	'.iRaw 			:=	TIIB[K4S8_DRL_03_E23_EL3314]^TC Inputs Channel 1^Value;
                                 .bError  		:=	TIIB[K4S8_DRL_03_E23_EL3314]^TC Inputs Channel 1^Error;
                                 .bUnderrange 	:=	TIIB[K4S8_DRL_03_E23_EL3314]^TC Inputs Channel 1^Underrange;
                                 .bOverrange  	:=	TIIB[K4S8_DRL_03_E23_EL3314]^TC Inputs Channel 1^Overrange
    '}
    {attribute 'pytmc' := ' pv: DREAM:STC:05'}
    TC_05 : FB_TempSensor;

    {attribute 'TcLinkTo' := 	'.iRaw 			:=	TIIB[K4S8_DRL_03_E23_EL3314]^TC Inputs Channel 2^Value;
                                 .bError  		:=	TIIB[K4S8_DRL_03_E23_EL3314]^TC Inputs Channel 2^Status^Error;
                                 .bUnderrange 	:=	TIIB[K4S8_DRL_03_E23_EL3314]^TC Inputs Channel 2^Status^Underrange;
                                 .bOverrange  	:=	TIIB[K4S8_DRL_03_E23_EL3314]^TC Inputs Channel 2^Status^Overrange
    '}
    {attribute 'pytmc' := ' pv: DREAM:STC:06'}
    TC_06 : FB_TempSensor;

    {attribute 'TcLinkTo' := 	'.iRaw 			:=	TIIB[K4S8_DRL_03_E23_EL3314]^TC Inputs Channel 3^Value;
                                 .bError  		:=	TIIB[K4S8_DRL_03_E23_EL3314]^TC Inputs Channel 3^Status^Error;
                                 .bUnderrange 	:=	TIIB[K4S8_DRL_03_E23_EL3314]^TC Inputs Channel 3^Status^Underrange;
                                 .bOverrange  	:=	TIIB[K4S8_DRL_03_E23_EL3314]^TC Inputs Channel 3^Status^Overrange
    '}
    {attribute 'pytmc' := ' pv: DREAM:STC:07'}
    TC_07 : FB_TempSensor;

    {attribute 'TcLinkTo' := 	'.iRaw 			:=	TIIB[K4S8_DRL_03_E23_EL3314]^TC Inputs Channel 4^Value;
                                 .bError  		:=	TIIB[K4S8_DRL_03_E23_EL3314]^TC Inputs Channel 4^Status^Error;
                                 .bUnderrange 	:=	TIIB[K4S8_DRL_03_E23_EL3314]^TC Inputs Channel 4^Status^Underrange;
                                 .bOverrange  	:=	TIIB[K4S8_DRL_03_E23_EL3314]^TC Inputs Channel 4^Status^Overrange
    '}
    {attribute 'pytmc' := ' pv: DREAM:STC:08'}
    TC_08 : FB_TempSensor;
END_VAR

// ---- GVLs/GVL_VAC_GAUGES.TcGVL
//{attribute 'qualified_only'}
VAR_GLOBAL
    (*Nozzle Chamber GPI*)
    {attribute 'pytmc' :=' pv: DREAM:NC:GPI:01'}
    {attribute 'TcLinkTo' := 	'.i_iPRESS_R	:=	TIIB[K4S8_DRL_03_E6_EL3174-0002]^AI Standard Channel 1^Value'}
    DREAM_NC_GPI_01 : FB_CVM201;

    {attribute 'TcLinkTo' := 	'.i_iPRESS_R		:=	TIIB[K4S8_DRL_03_E5_EL3174-0002]^AI Standard Channel 1^Value;
                                 .i_xHV_ON			:=	TIIB[K4S8_DRL_03_E4_EL1084]^Channel 3^Input;
                                 .q_xHV_DIS			:=	TIIB[K4S8_DRL_03_E1_EL2624]^Channel 1^Output
    '}

    (*Nozzle Chamber GCC*)
    {attribute 'pytmc' :=' pv: DREAM:NC:GCC:01'}
    DREAM_NC_GCC_01: FB_CCM501;

    (*DP1 GHC*)
    {attribute 'TcLinkTo' := 	'.i_iPRESS_R		:=	TIIB[K4S8_DRL_03_E5_EL3174-0002]^AI Standard Channel 2^Value;
                                 .i_xHV_ON			:=	TIIB[K4S8_DRL_03_E4_EL1084]^Channel 4^Input;
                                 .q_xHV_DIS			:=	TIIB[K4S8_DRL_03_E1_EL2624]^Channel 2^Output
    '}
    {attribute 'pytmc' :=' pv: DREAM:DP1:GHC:01'}
    DREAM_DP1_GHC_01 : FB_IMG401;

    (*DP1 GPI*)
    {attribute 'pytmc' :=' pv: DREAM:DP1:GPI:01'}
    {attribute 'TcLinkTo' := 	'.i_iPRESS_R	:=	TIIB[K4S8_DRL_03_E6_EL3174-0002]^AI Standard Channel 2^Value'}
    DREAM_DP1_GPI_01 : FB_CVM201;

    (*DP2 GHC*)
    {attribute 'TcLinkTo' := 	'.i_iPRESS_R		:=	TIIB[K4S8_DRL_03_E5_EL3174-0002]^AI Standard Channel 3^Value;
                                 .i_xHV_ON			:=	TIIB[K4S8_DRL_03_E4_EL1084]^Channel 1^Input;
                                 .q_xHV_DIS			:=	TIIB[K4S8_DRL_03_E1_EL2624]^Channel 3^Output
    '}
    {attribute 'pytmc' :=' pv: DREAM:DP2:GHC:01'}
    DREAM_DP2_GHC_01 : FB_IMG401;

    (*DP3 GHC*)
    {attribute 'TcLinkTo' := 	'.i_iPRESS_R		:=	TIIB[K4S8_DRL_03_E5_EL3174-0002]^AI Standard Channel 4^Value;
                                 .i_xHV_ON			:=	TIIB[K4S8_DRL_03_E4_EL1084]^Channel 2^Input;
                                 .q_xHV_DIS			:=	TIIB[K4S8_DRL_03_E1_EL2624]^Channel 4^Output
    '}
    {attribute 'pytmc' :=' pv: DREAM:DP3:GHC:01'}
    DREAM_DP3_GHC_01 : FB_IMG401;

    (*MC HOT CATHODE GUAGE*)
    {attribute 'TcLinkTo' := 	'.i_iPRESS_R_CH1	:=	TIIB[R03_DRL_01_E3_EL3174-0002]^AI Standard Channel 1^Value;
                                 .i_iPRESS_R_CH2	:=	TIIB[R03_DRL_01_E3_EL3174-0002]^AI Standard Channel 2^Value;
                                 .i_xHV_ON			:=	TIIB[R03_DRL_01_E1_EL1004]^Channel 1^Input;
                                 .i_xCH2_SEL		:=	TIIB[R03_DRL_01_E1_EL1004]^Channel 2^Input;
                                 .i_xERR_CH1		:=	TIIB[R03_DRL_01_E1_EL1004]^Channel 3^Input;
                                 .i_xERR_CH2		:=	TIIB[R03_DRL_01_E1_EL1004]^Channel 4^Input;
                                 .q_xHV_DIS_CH1		:=	TIIB[R03_DRL_01_E2_EL2624]^Channel 1^Output;
                                 .q_xHV_DIS_CH2		:=	TIIB[R03_DRL_01_E2_EL2624]^Channel 2^Output
    '}
    {attribute 'pytmc' :=' pv: DREAM:MC:GHC'}
    DREAM_MC_GHC : FB_IE514;

    //main chamber global gauge structure - updated based on hot cahtode is selected or use pirani if both hot cathode gauges are off
    {attribute 'pytmc' :=' pv: DREAM:MC:GAUGE:01'}
    stDREAM_MC_GAUGE : ST_VG;

    //main chamber GHC gauge structure - updated based on which channel selected in the leybold hot cathode gauge
    {attribute 'pytmc' :=' pv: DREAM:MC:GHC:GAUGE:01'}
    stDREAM_MC_GHC_GAUGE : ST_VG;

    //CAT1 chamber global gauge structure - updated based on  hot cahtode is selected or use pirani if both hot cathode gauges are off
    {attribute 'pytmc' :=' pv: DREAM:CAT1:GAUGE:01'}
    stDREAM_CAT1_GAUGE : ST_VG;

    (*MC GPI*)
    {attribute 'TcLinkTo' := 	'.i_iPRESS_R	:=	TIIB[K4S8_DRL_04_E16_EL3174-0002]^AI Standard Channel 1^Value'}
    {attribute 'pytmc' := 'pv: DREAM:MC:GPI:01'}
    DREAM_MC_GPI_01 : FB_MKS275;

    (*CATCHER 1*)
    {attribute 'TcLinkTo' := 	'    .i_iPRESS_R		:=	TIIB[K4S8_DRL_04_E16_EL3174-0002]^AI Standard Channel 2^Value;
                                     .i_xHV_ON			:=	TIIB[K4S8_DRL_04_E15_EL1084]^Channel 1^Input;
                                     .q_xHV_DIS			:=	TIIB[K4S8_DRL_04_E14_EL2624]^Channel 1^Output
    '}
    {attribute 'pytmc' :=' pv: DREAM:CAT1:GHC:01'}
    DREAM_CAT1_GHC_01 : FB_IMG401;

    (*CATCHER 2*)
    {attribute 'TcLinkTo' := 	'    .i_iPRESS_R		:=	TIIB[K4S8_DRL_04_E16_EL3174-0002]^AI Standard Channel 3^Value;
                                     .i_xHV_ON			:=	TIIB[K4S8_DRL_04_E15_EL1084]^Channel 2^Input;
                                     .q_xHV_DIS			:=	TIIB[K4S8_DRL_04_E14_EL2624]^Channel 2^Output
    '}
    {attribute 'pytmc' :=' pv: DREAM:CAT2:GHC:01'}
    DREAM_CAT2_GHC_01 : FB_IMG401;

    (*ROUGHING PIRANIs*)
    //Micro piranis 925
    {attribute 'TcLinkTo' := 	'.i_iPRESS_R	:=	TIIB[WALL_E_PPL_01_EP1_EP4374-0002]^AI Inputs Channel 1^Value'}
    {attribute 'pytmc' := 'pv: DREAM:ROUGH1:GPI:01'}
    DREAM_ROUGH1_GPI_01 : FB_9XX;

    {attribute 'TcLinkTo' := 	'.i_iPRESS_R	:=	TIIB[K4S8_DRL_04_EP1_EP4374-0002]^AI Inputs Channel 1^Value'}
    {attribute 'pytmc' := 'pv: DREAM:ROUGH1:GPI:02'}
    DREAM_ROUGH1_GPI_02 : FB_9XX;

    {attribute 'TcLinkTo' := 	'.i_iPRESS_R	:=	TIIB[WALL_E_PPL_01_EP1_EP4374-0002]^AI Inputs Channel 2^Value'}
    {attribute 'pytmc' := 'pv: DREAM:ROUGH2:GPI:01'}
    DREAM_ROUGH2_GPI_01 : FB_9XX;

    {attribute 'TcLinkTo' := 	'.i_iPRESS_R	:=	TIIB[K4S8_DRL_04_EP1_EP4374-0002]^AI Inputs Channel 2^Value'}
    {attribute 'pytmc' := 'pv: DREAM:ROUGH2:GPI:02'}
    DREAM_ROUGH2_GPI_02 : FB_9XX;

    {attribute 'TcLinkTo' := 	'.i_iPRESS_R	:=	TIIB[K4S8_DRL_04_EP2_EP4374-0002]^AI Inputs Channel 1^Value'}
    {attribute 'pytmc' := 'pv: DREAM:ROUGH2:GPI:03'}
    DREAM_ROUGH2_GPI_03 : FB_9XX;

END_VAR

// ---- GVLs/GVL_VAC_PUMPS.TcGVL
//{attribute 'qualified_only'}
VAR_GLOBAL
    (*NOZZLE CHAMBER*)
    {attribute 'TcLinkTo' := 	'.i_xAtSpd			:=	TIIB[K4S8_DRL_03_E13_EL1004]^Channel 1^Input;
                                 .i_xFaultNC		:=	TIIB[K4S8_DRL_03_E13_EL1004]^Channel 3^Input;
                                 .i_xRemote         :=  TIIB[K4S8_DRL_03_E13_EL1004]^Channel 2^Input;
                                 .q_RunDO			:=	TIIB[K4S8_DRL_03_E14_EL2004]^Channel 1^Output;
                                 .q_PumpingStation  :=	TIIB[K4S8_DRL_03_E14_EL2004]^Channel 3^Output;
                                 .q_xRemote	        :=	TIIB[K4S8_DRL_03_E14_EL2004]^Channel 2^Output
     '}
     {attribute 'pytmc' :=' pv: DREAM:NC:PTM:01'}
     DREAM_NC_PTM_01 : FB_PTM_Pfeiffer;

     {attribute 'TcLinkTo' := 	'.i_xAtSpd			:=	TIIB[K4S8_DRL_03_E16_EL1004]^Channel 1^Input;
                                 .i_xFaultNC		:=	TIIB[K4S8_DRL_03_E16_EL1004]^Channel 3^Input;
                                 .i_xRemote         :=  TIIB[K4S8_DRL_03_E16_EL1004]^Channel 2^Input;
                                 .q_RunDO			:=	TIIB[K4S8_DRL_03_E17_EL2004]^Channel 1^Output;
                                 .q_PumpingStation  :=	TIIB[K4S8_DRL_03_E17_EL2004]^Channel 3^Output;
                                 .q_xRemote	        :=	TIIB[K4S8_DRL_03_E17_EL2004]^Channel 2^Output
    '}
    {attribute 'pytmc' :=' pv: DREAM:NC:PTM:02'}
    DREAM_NC_PTM_02 : FB_PTM_Pfeiffer;

    (*DP1*)
    {attribute 'TcLinkTo' := 	'.i_xAtSpd			:=	TIIB[K4S8_DRL_03_E19_EL1004]^Channel 1^Input;
                                 .i_xFaultNC		:=	TIIB[K4S8_DRL_03_E19_EL1004]^Channel 3^Input;
                                 .i_xRemote         :=  TIIB[K4S8_DRL_03_E19_EL1004]^Channel 2^Input;
                                 .q_RunDO			:=	TIIB[K4S8_DRL_03_E20_EL2004]^Channel 1^Output;
                                 .q_PumpingStation  :=	TIIB[K4S8_DRL_03_E20_EL2004]^Channel 3^Output;
                                 .q_xRemote	        :=	TIIB[K4S8_DRL_03_E20_EL2004]^Channel 2^Output
    '}
    {attribute 'pytmc' :=' pv: DREAM:DP1:PTM:01'}
    DREAM_DP1_PTM_01 : FB_PTM_Pfeiffer;

    (*DP2*)
    {attribute 'TcLinkTo' := 	'.i_xAtSpd			:=	TIIB[R20_DRL_03_E4_EL1004]^Channel 2^Input;
                                 .i_xFaultNC		:=	TIIB[R20_DRL_03_E4_EL1004]^Channel 1^Input;
                                 .q_RunDO			:=	TIIB[R20_DRL_03_E7_EL2794]^Channel 1^Output
     '}
    {attribute 'pytmc' :=' pv: DREAM:DP2:PTM:01'}
    DREAM_DP2_PTM_01 : FB_PTM_TurboDrive;

    (*DP3*)
    {attribute 'TcLinkTo' := 	'.i_xAtSpd			:=	TIIB[R20_DRL_03_E4_EL1004]^Channel 4^Input;
                                 .i_xFaultNC		:=	TIIB[R20_DRL_03_E4_EL1004]^Channel 3^Input;
                                 .q_RunDO			:=	TIIB[R20_DRL_03_E7_EL2794]^Channel 3^Output
    '}
    {attribute 'pytmc' :=' pv: DREAM:DP3:PTM:01'}
    DREAM_DP3_PTM_01 : FB_PTM_TurboDrive;


    (*MAIN CHAMBER*)
    {attribute 'TcLinkTo' := 	'.i_xAtSpd			:=	TIIB[R20_DRL_03_E5_EL1004]^Channel 2^Input;
                                 .i_xFaultNC		:=	TIIB[R20_DRL_03_E5_EL1004]^Channel 1^Input;
                                 .q_RunDO			:=	TIIB[R20_DRL_03_E7_EL2794]^Channel 2^Output
    '}
    {attribute 'pytmc' :=' pv: DREAM:MC:PTM:01'}
    DREAM_MC_PTM_01 : FB_PTM_TurboDrive;

    {attribute 'TcLinkTo' := 	'.i_xAtSpd			:=	TIIB[R20_DRL_03_E5_EL1004]^Channel 4^Input;
                                 .i_xFaultNC		:=	TIIB[R20_DRL_03_E5_EL1004]^Channel 3^Input;
                                 .q_RunDO			:=	TIIB[R20_DRL_03_E7_EL2794]^Channel 4^Output
    '}
    {attribute 'pytmc' :=' pv: DREAM:MC:PTM:02'}
    DREAM_MC_PTM_02 : FB_PTM_TurboDrive;

    (*BOOSTER TURBO PUMPS ROUGHING*)
    {attribute 'TcLinkTo' := 	'.i_xAtSpd			:=	TIIB[K4S8_DRL_04_E3_EL1004]^Channel 2^Input;
                                 .i_xFaultNC		:=	TIIB[K4S8_DRL_04_E3_EL1004]^Channel 1^Input;
                                 .q_RunDO			:=	TIIB[K4S8_DRL_04_E5_EL2794]^Channel 1^Output
    '}
    {attribute 'pytmc' :=' pv: DREAM:ROUGH2:PTM:01'}
    DREAM_ROUGH2_PTM_01 : FB_PTM_TurboDrive;

    {attribute 'TcLinkTo' := 	'.i_xAtSpd			:=	TIIB[K4S8_DRL_04_E4_EL1004]^Channel 4^Input;
                                 .i_xFaultNC		:=	TIIB[K4S8_DRL_04_E4_EL1004]^Channel 3^Input;
                                 .q_RunDO			:=	TIIB[K4S8_DRL_04_E5_EL2794]^Channel 4^Output
    '}
    {attribute 'pytmc' :=' pv: DREAM:ROUGH2:PTM:02'}
    DREAM_ROUGH2_PTM_02 : FB_PTM_TurboDrive;

    (*CATCHER 1*)
    {attribute 'TcLinkTo' := 	'.i_xAtSpd			:=	TIIB[K4S8_DRL_04_E3_EL1004]^Channel 4^Input;
                                 .i_xFaultNC		:=	TIIB[K4S8_DRL_04_E3_EL1004]^Channel 3^Input;
                                 .q_RunDO			:=	TIIB[K4S8_DRL_04_E5_EL2794]^Channel 2^Output
    '}
    {attribute 'pytmc' :=' pv: DREAM:CAT1:PTM:01'}
    DREAM_CAT1_PTM_01 : FB_PTM_TurboDrive;

    (*CATCHER 2*)
    {attribute 'TcLinkTo' := 	'.i_xAtSpd			:=	TIIB[K4S8_DRL_04_E4_EL1004]^Channel 2^Input;
                                 .i_xFaultNC		:=	TIIB[K4S8_DRL_04_E4_EL1004]^Channel 1^Input;
                                 .q_RunDO			:=	TIIB[K4S8_DRL_04_E5_EL2794]^Channel 3^Output
    '}
    {attribute 'pytmc' :=' pv: DREAM:CAT2:PTM:01'}
    DREAM_CAT2_PTM_01 : FB_PTM_TurboDrive;

    //Turbo Pumps Running evaluation bit
    bMCPumpsRunning : BOOL;
    bCATPumpsRunning : BOOL;


    (*Serial Interface*)
    (*Pfeiffer TC400 serial*)
    stPfeiffer_CTRL_DREAM_NC_PTM_01  : ARRAY[1..gcMaxPfeifferPumps] OF ST_PfeifferControl;
    stPfeiffer_RBK_DREAM_NC_PTM_01   : ARRAY[1..gcMaxPfeifferPumps] OF ST_PfeifferStatus;
    fbPfeifferCom_DREAM_NC_PTM_01    : FB_PFEIFFER_COM;

    stPfeiffer_CTRL_DREAM_NC_PTM_02  : ARRAY[1..gcMaxPfeifferPumps] OF ST_PfeifferControl;
    stPfeiffer_RBK_DREAM_NC_PTM_02   : ARRAY[1..gcMaxPfeifferPumps] OF ST_PfeifferStatus;
    fbPfeifferCom_DREAM_NC_PTM_02    : FB_PFEIFFER_COM;

    stPfeiffer_CTRL_DREAM_DP1_PTM_01 : ARRAY[1..gcMaxPfeifferPumps] OF ST_PfeifferControl;
    stPfeiffer_RBK_DREAM_DP1_PTM_01	 : ARRAY[1..gcMaxPfeifferPumps] OF ST_PfeifferStatus;
    fbPfeifferCom_DREAM_DP1_PTM_01   : FB_PFEIFFER_COM;

    (*Leybold TD20 serial*)
    stTD20_RBK_DREAM_DP2_PTM_01      : ST_TD20Status;
    fbTD20Com_DREAM_DP2_PTM_01       : FB_OERLIKON_TD20_COM;

    stTD20_RBK_DREAM_DP3_PTM_01      : ST_TD20Status;
    fbTD20Com_DREAM_DP3_PTM_01       : FB_OERLIKON_TD20_COM;

    stTD20_RBK_DREAM_MC_PTM_01       : ST_TD20Status;
    fbTD20Com_DREAM_MC_PTM_01        : FB_OERLIKON_TD20_COM;

    stTD20_RBK_DREAM_MC_PTM_02       : ST_TD20Status;
    fbTD20Com_DREAM_MC_PTM_02        : FB_OERLIKON_TD20_COM;

    (*Leybold TD400 serial*)
    stTD400_RBK_DREAM_CAT1_PTM_01    : ST_TD400Status;
    stTD400_CTRL_DREAM_CAT1_PTM_01   : ST_TD400Control;
    fbTD400Com_DREAM_CAT1_PTM_01     : FB_OERLIKON_TD400_COM;
    fbTD400SerialIO_DREAM_CAT1_PTM_01: FB_OERLIKON_TD400_TO_PTM;

    stTD400_RBK_DREAM_CAT2_PTM_01    : ST_TD400Status;
    stTD400_CTRL_DREAM_CAT2_PTM_01   : ST_TD400Control;
    fbTD400Com_DREAM_CAT2_PTM_01     : FB_OERLIKON_TD400_COM;
    fbTD400SerialIO_DREAM_CAT2_PTM_01: FB_OERLIKON_TD400_TO_PTM;

    stTD400_RBK_DREAM_ROUGH2_PTM_01  : ST_TD400Status;
    stTD400_CTRL_DREAM_ROUGH2_PTM_01 : ST_TD400Control;
    fbTD400Com_DREAM_ROUGH2_PTM_01   : FB_OERLIKON_TD400_COM;
    fbTD400SerialIO_DREAM_ROUGH2_PTM_01: FB_OERLIKON_TD400_TO_PTM;

    stTD400_RBK_DREAM_ROUGH2_PTM_02  : ST_TD400Status;
    stTD400_CTRL_DREAM_ROUGH2_PTM_02 : ST_TD400Control;
    fbTD400Com_DREAM_ROUGH2_PTM_02   : FB_OERLIKON_TD400_COM;
    fbTD400SerialIO_DREAM_ROUGH2_PTM_02: FB_OERLIKON_TD400_TO_PTM;

END_VAR

// ---- GVLs/GVL_VAC_VALVES.TcGVL
//{attribute 'qualified_only'}
VAR_GLOBAL
    (*DP1 ISOLATION VALVE*)
    {attribute 'TcLinkTo' := 	'.i_xOpnLS	:=	TIIB[K4S8_DRL_03_E10_EL1004]^Channel 1^Input;
                                 .i_xClsLS	:=	TIIB[K4S8_DRL_03_E10_EL1004]^Channel 2^Input;
                                 .q_xOPN_DO	:=	TIIB[K4S8_DRL_03_E11_EL2004]^Channel 2^Output
    '}
    {attribute 'pytmc' :=' pv: DREAM:DP1:VRC:01'}
    DREAM_DP1_VRC_01: FB_VGC;

    {attribute 'TcLinkTo' := 	'.i_xOpnLS	:=	TIIB[K4S8_DRL_03_E10_EL1004]^Channel 3^Input;
                                 .i_xClsLS	:=	TIIB[K4S8_DRL_03_E10_EL1004]^Channel 4^Input;
                                 .q_xCLS_DO	:=	TIIB[K4S8_DRL_03_E11_EL2004]^Channel 1^Output
    '}
    {attribute 'pytmc' :=' pv: DREAM:DP1:VRC:02'}
    DREAM_DP1_VRC_02: FB_VRC_NO;

    (*Test dual-acting valve, no interlock implemented, contact Tong*)
    {attribute 'TcLinkTo' := 	'.i_xOpnLS	:=	TIIB[K4S8_DRL_04_E1_EL1004]^Channel 3^Input;
                                 .i_xClsLS	:=	TIIB[K4S8_DRL_04_E1_EL1004]^Channel 4^Input;
                                 .q_xOPN_DO	:=	TIIB[K4S8_DRL_04_E2_EL2004]^Channel 3^Output;
                                 .q_xCLS_DO	:=	TIIB[K4S8_DRL_04_E2_EL2004]^Channel 4^Output



    '}
    {attribute 'pytmc' :=' pv: DREAM:DP1:VRC:20'}
    DREAM_DP1_VRC_20: FB_VRC_DA;

    (*CATCHER 1 ISOLATION VALVE*)
    {attribute 'TcLinkTo' := 	'.i_xOpnLS	:=	TIIB[K4S8_DRL_04_E1_EL1004]^Channel 1^Input;
                                 .i_xClsLS	:=	TIIB[K4S8_DRL_04_E1_EL1004]^Channel 2^Input;
                                 .q_xOPN_DO	:=	TIIB[K4S8_DRL_04_E2_EL2004]^Channel 1^Output
    '}
    {attribute 'pytmc' :=' pv: DREAM:CAT1:VRC:01'}
    DREAM_CAT1_VRC_01: FB_VGC;

    (*ANGLE VALVES ROUGHING*)
    //Pneumatic valves
    {attribute 'TcLinkTo' := 	'.i_xOpnLS	:=	TIIB[K4S8_DRL_04_E9_EL1004]^Channel 1^Input;
                                 .i_xClsLS	:=	TIIB[K4S8_DRL_04_E9_EL1004]^Channel 2^Input;
                                 .q_xOPN_DO	:=	TIIB[K4S8_DRL_04_E11_EL2004]^Channel 1^Output
    '}
    {attribute 'pytmc' :=' pv: DREAM:ROUGH1:VRC:01'}
    DREAM_ROUGH1_VRC_01: FB_VGC;

    {attribute 'TcLinkTo' := 	'.i_xOpnLS	:=	TIIB[K4S8_DRL_04_E9_EL1004]^Channel 3^Input;
                                 .i_xClsLS	:=	TIIB[K4S8_DRL_04_E9_EL1004]^Channel 4^Input;
                                 .q_xOPN_DO	:=	TIIB[K4S8_DRL_04_E11_EL2004]^Channel 2^Output
    '}
    {attribute 'pytmc' :=' pv: DREAM:ROUGH2:VRC:01'}
    DREAM_ROUGH2_VRC_01: FB_VGC;

    {attribute 'TcLinkTo' := 	'.i_xOpnLS	:=	TIIB[K4S8_DRL_04_E10_EL1004]^Channel 1^Input;
                                 .i_xClsLS	:=	TIIB[K4S8_DRL_04_E10_EL1004]^Channel 2^Input;
                                 .q_xOPN_DO	:=	TIIB[K4S8_DRL_04_E11_EL2004]^Channel 3^Output
    '}
    {attribute 'pytmc' :=' pv: DREAM:ROUGH2:VRC:02'}
    DREAM_ROUGH2_VRC_02: FB_VGC;

    {attribute 'TcLinkTo' := 	'.i_xOpnLS	:=	TIIB[K4S8_DRL_04_E10_EL1004]^Channel 3^Input;
                                 .i_xClsLS	:=	TIIB[K4S8_DRL_04_E10_EL1004]^Channel 4^Input;
                                 .q_xOPN_DO	:=	TIIB[K4S8_DRL_04_E11_EL2004]^Channel 4^Output
    '}

    //valve added tempfor testing only
   {attribute 'pytmc' :=' pv: DREAM:ROUGH1:VRC:20'}
    DREAM_ROUGH1_VRC_20: FB_VRC;

    //Manifold roughing valve
    {attribute 'TcLinkTo' := 	'.i_xOpnLS	:=	TIIB[WALL_E_PPL_01_EP2_EP2338-0002]^Channel 1^Input;
                                 .i_xClsLS	:=	TIIB[WALL_E_PPL_01_EP2_EP2338-0002]^Channel 2^Input;
                                 .q_xOPN_DO	:=	TIIB[WALL_E_PPL_01_EP2_EP2338-0002]^Channel 11^Output
    '}
    {attribute 'pytmc' :=' pv: DREAM:ROUGH1:VRC:10'}
    DREAM_ROUGH1_VRC_10: FB_VRC;

    (*VENT VALVES ROUGHING*)
    //FLow Control valves MKS248
    {attribute 'TcLinkTo' := 	'.q_iRawPosition	:=	TIIB[WALL_E_PPL_01_EP1_EP4374-0002]^AO Outputs Channel 3^Analog output'}
    {attribute 'pytmc' := 'pv: DREAM:ROUGH1:VFV:01'}
    DREAM_ROUGH1_VFV_01 : FB_MKS248;

    {attribute 'TcLinkTo' := 	'.q_iRawPosition	:=	TIIB[K4S8_DRL_04_EP1_EP4374-0002]^AO Outputs Channel 3^Analog output'}
    {attribute 'pytmc' := 'pv: DREAM:ROUGH1:VFV:02'}
    DREAM_ROUGH1_VFV_02 : FB_MKS248;

    {attribute 'TcLinkTo' := 	'.q_iRawPosition	:=	TIIB[WALL_E_PPL_01_EP1_EP4374-0002]^AO Outputs Channel 4^Analog output'}
    {attribute 'pytmc' := 'pv: DREAM:ROUGH2:VFV:01'}
    DREAM_ROUGH2_VFV_01 : FB_MKS248;

    {attribute 'TcLinkTo' := 	'.q_iRawPosition	:=	TIIB[K4S8_DRL_04_EP1_EP4374-0002]^AO Outputs Channel 4^Analog output'}
    {attribute 'pytmc' := 'pv: DREAM:ROUGH2:VFV:02'}
    DREAM_ROUGH2_VFV_02 : FB_MKS248;

    {attribute 'TcLinkTo' := 	'.q_iRawPosition	:=	TIIB[K4S8_DRL_04_EP2_EP4374-0002]^AO Outputs Channel 3^Analog output'}
    {attribute 'pytmc' := 'pv: DREAM:ROUGH2:VFV:03'}
    DREAM_ROUGH2_VFV_03 : FB_MKS248;

END_VAR

// ---- GVLs/GVL_Variables.TcGVL
//{attribute 'qualified_only'}
VAR_GLOBAL
    {attribute 'pytmc' := '
        pv: PLC:DREAM:VAC:OVRDON
        io: io
    '}
    bSystemOverrideMode	: BOOL := FALSE; (* Global system override for the DREAM Vacuum System*)

    {attribute 'pytmc' := '
        pv: PLC:DREAM:ON_BEAMLINE
        io: i
    '}
    bOnBeamline	: BOOL := FALSE;

    //HV Interlock Pressure setpoint default is 1e-5 Torr, when switched to MC pirani gauge this value will change to 5e-04 Torr.
    {attribute 'pytmc' := '
        pv: PLC:DREAM:HV_MAX_PRESS_SP
        io: io
    '}
    fHighVoltageMaxPressure : REAL := 1e-05; (*inital High voltage Minimum Enable Pressure*)

     {attribute 'pytmc' := '
    pv: HV:GPI:SP;
    io:io;
    field: HOPR 1000
    field: LOPR 0
    field: PREC 2
    field: EGU "TORR"
    autosave_pass1: VAL DESC
    '}
    rHV_GPI_SP: REAL := 0.0005; (*inital high voltage setpoint *)

END_VAR

// ---- POUs/MAIN.TcPOU
PROGRAM MAIN
VAR
    fbLogHandler : FB_LogHandler;
END_VAR

fbLogHandler();

PRG_ECAT_CHECK();

PRG_GAUGES();

PRG_VALVES();

PRG_TURBO_PUMPS();

PRG_HV_ILK();

PRG_COIL_PS_ILK();

PRG_TC();

END_PROGRAM

// ---- POUs/PRG_ECAT_CHECK.TcPOU
PROGRAM PRG_ECAT_CHECK
VAR
    //EtherCAT bridge error
    bEcatBridge_COM_ERROR : BOOL;

    //Ethercat bridge error for DREAM Motion
    bMotEcatBridge_COM_ERROR : BOOL;
END_VAR

(*EtherCAT Bridge Status*)
//bEcatBridge_COM_ERROR = TRUE means that there is an EtherCAT Bridge Communication Error.
bEcatBridge_COM_ERROR := (bEcatBridge_TxPDO_state OR bEcatBridge_External_device_not_connected OR bEcatBridge_WcState);

bOnBeamline := (bEcatBridge_COM_ERROR = FALSE) AND (sHUTCH_PLC_NAME = 'TMO');

bMotEcatBridge_COM_ERROR := (bMotEcatBridge_TxPDO_state OR bMotEcatBridge_External_device_not_connected OR bMotEcatBridge_WcState);

END_PROGRAM

// ---- POUs/PRG_GAUGES.TcPOU
PROGRAM PRG_GAUGES
VAR

END_VAR

(**Gas Injection Gauges**)
//Pirani MKS 275 Gauges
DREAM_NC_GPI_01.M_SetBits(30518);
DREAM_NC_GPI_01(PG=>);
DREAM_DP1_GPI_01.M_SetBits(30518);
DREAM_DP1_GPI_01(PG=>);

//Cold Cathode Guages
DREAM_NC_GCC_01.M_SetBits(30518);
DREAM_NC_GCC_01(PG:= DREAM_NC_GPI_01.PG);

//Hot Cathode Guages
DREAM_DP1_GHC_01.M_SetBits(30518);
DREAM_DP1_GHC_01(PG:= DREAM_DP1_GPI_01.PG, IG=>);
DREAM_DP2_GHC_01.M_SetBits(30518);
DREAM_DP2_GHC_01(PG:= DREAM_DP1_GPI_01.PG, IG=>);
DREAM_DP3_GHC_01.M_SetBits(30518);
DREAM_DP3_GHC_01(PG:= DREAM_DP1_GPI_01.PG, IG=>);

(**Main Chmamber Gauges**)
//Pirani Gauges
DREAM_MC_GPI_01.M_SetBits(30518);
DREAM_MC_GPI_01();

//Hot Cathode gauge IE514
DREAM_MC_GHC.M_SetBits(30518);
//Using DP3:GHC to interlock main chamber gauge because protetion setpoint for the gauge has to be set to 1e-6 - 1E-5
//Changing back to interlock MC HC gauge with MC pirani gauge, becasue when coil is ON it can turn OFF DP3 gauge which then affect interlocks for the beamline valves and catcher valve
DREAM_MC_GHC(PG:= DREAM_MC_GPI_01.PG); //This fb reads statuses and control two gauges DREAM:MC:GHC:01 and DREAM:MC:GHC:02

//Update stDREAM_MC_GHC_GAUGE structure based on CH selected by controller and data to TMO Beamline Vacuum PLC
IF DREAM_MC_GHC.M_IsCh1Selected() THEN
    stDREAM_MC_GHC_GAUGE := DREAM_MC_GHC.IG_CH1;

    GVL_PLC_Interface.bDREAM_MAIN_xAT_VAC := DREAM_MC_GHC.IG_CH1.xAT_VAC;
    GVL_PLC_Interface.bDREAM_MAIN_xPRESS_OK := DREAM_MC_GHC.IG_CH1.xPRESS_OK;
    GVL_PLC_Interface.fDREAM_MAIN_rPRESS := DREAM_MC_GHC.IG_CH1.rPRESS;

ELSIF DREAM_MC_GHC.M_IsCh2Selected() THEN
    stDREAM_MC_GHC_GAUGE := DREAM_MC_GHC.IG_CH2;

    GVL_PLC_Interface.bDREAM_MAIN_xAT_VAC := DREAM_MC_GHC.IG_CH2.xAT_VAC;
    GVL_PLC_Interface.bDREAM_MAIN_xPRESS_OK := DREAM_MC_GHC.IG_CH2.xPRESS_OK;
    GVL_PLC_Interface.fDREAM_MAIN_rPRESS := DREAM_MC_GHC.IG_CH2.rPRESS;
END_IF

//Switch to Pirani gauge, when High vacuum gauge is not available, check pumps running when using Pirani
IF NOT stDREAM_MC_GHC_GAUGE.xPRESS_OK THEN
//This interlock pseudo MC gauge is also assigned in the PRG_Valves, it is redanduncy and make sure change the PRG_Valves as well if change here
    stDREAM_MC_GAUGE := DREAM_MC_GPI_01.PG;
    GVL_PLC_Interface.bDREAM_MAIN_xAT_VAC := DREAM_MC_GPI_01.PG.xAT_VAC;
    GVL_PLC_Interface.bDREAM_MAIN_xPRESS_OK := DREAM_MC_GPI_01.PG.xPRESS_OK AND bMCPumpsRunning;
    GVL_PLC_Interface.fDREAM_MAIN_rPRESS := DREAM_MC_GPI_01.PG.rPRESS;
ElSE
//This interlock pseudo MC gauge is also assigned in the PRG_Valves, it is redanduncy and make sure change the PRG_Valves as well if change here
    stDREAM_MC_GAUGE := stDREAM_MC_GHC_GAUGE;
    GVL_PLC_Interface.bDREAM_MAIN_xAT_VAC := stDREAM_MC_GHC_GAUGE.xAT_VAC;
    GVL_PLC_Interface.bDREAM_MAIN_xPRESS_OK := stDREAM_MC_GHC_GAUGE.xPRESS_OK;
    GVL_PLC_Interface.fDREAM_MAIN_rPRESS := stDREAM_MC_GHC_GAUGE.rPRESS;
END_IF



(**Catcher Gauges**)
//Hot Cathode Guages
DREAM_CAT1_GHC_01.M_SetBits(30518);
DREAM_CAT1_GHC_01(PG:= DREAM_ROUGH2_GPI_03.PG);
DREAM_CAT2_GHC_01.M_SetBits(30518);
DREAM_CAT2_GHC_01(PG:= DREAM_ROUGH2_GPI_03.PG);

(**Roughing Section Gauges**)
DREAM_ROUGH1_GPI_01.M_SetBits(32767);
DREAM_ROUGH1_GPI_01();
DREAM_ROUGH1_GPI_02.M_SetBits(32767);
DREAM_ROUGH1_GPI_02();

DREAM_ROUGH2_GPI_01.M_SetBits(32767);
DREAM_ROUGH2_GPI_01();
DREAM_ROUGH2_GPI_02.M_SetBits(32767);
DREAM_ROUGH2_GPI_02();
DREAM_ROUGH2_GPI_03.M_SetBits(32767);
DREAM_ROUGH2_GPI_03();

END_PROGRAM

// ---- POUs/PRG_VALVES.TcPOU
PROGRAM PRG_VALVES
VAR
    //Rough lines VRC external interlocks
    bROUGH1_VRC_01_ILK : BOOL;
    bROUGH2_VRC_01_ILK : BOOL;
    bROUGH2_VRC_02_ILK : BOOL;
    bROUGH1_VRC_01_Override : BOOL;
    bROUGH2_VRC_01_Override : BOOL;
    bROUGH2_VRC_02_Override : BOOL;
    bCAT1_VRC_01_ExtILK : BOOL;
    bDP1_VRC_01_ILK : BOOL;
    bDP1_VRC_02_ILK : BOOL;
    bCAT1_VRC_01_ExtILK_US:BOOL;
    bCAT1_VRC_01_ExtILK_DS:BOOL;
    bCAT1_DisableDiffIlk : BOOL;

    //dummy FF output to use in VGC_2S function
    dummy_FFFO : FB_HardwareFFOutput;
    dummy_fbArbiter1 : FB_Arbiter(1);
END_VAR

(**Gas Injection Valves**)
DREAM_DP1_VRC_01(i_stUSG := DREAM_NC_GPI_01.PG,
                 i_stDSG := DREAM_DP1_GPI_01.PG,
                 i_xDis_DPIlk := FALSE,
                 i_xEPS_OK := TRUE,
                 i_xPMPS_OK := TRUE,
                 i_xReset := FALSE,
                 i_xExt_OK := TRUE,
                 i_xOverrideMode := bSystemOverrideMode,
                 io_fbFFHWO := dummy_FFFO,
                 fbArbiter := dummy_fbArbiter1,
                 i_sDevName := 'DREAM-DP1-VRC-01');

//DP1_VRC_02 Interlock evaluation NOTE: Normally OPEN Valve!!
bDP1_VRC_02_ILK := DREAM_DP1_VRC_01.iq_stValve.i_xOpnLS; //Interlock changed for this valve to only gets interlocked by DREAM_DP1_VRC_01 valve

DREAM_DP1_VRC_02(i_xExtILK_OK := bDP1_VRC_02_ILK, i_xOverrideMode := bSystemOverrideMode); //Normally open valve

(**Catcher valve**)

//CAT1_VRC_01 Interlock evaluation
//Select US interlock gauge and adding pump running interlock when use Pirani
IF NOT stDREAM_MC_GHC_GAUGE.xPRESS_OK THEN
    bCAT1_VRC_01_ExtILK_US := bMCPumpsRunning;
//This interlock pseudo gauge is also assigned in the PRG_Gauge, it is redanduncy and make sure change the PRG_Gauge as well if change here
    stDREAM_MC_GAUGE := DREAM_MC_GPI_01.PG;
    stDREAM_MC_GAUGE.sPath := 'DREAM_MC_GPI_01';
ELSE
    bCAT1_VRC_01_ExtILK_US := True;
//This interlock pseudo MC gauge is also assigned in the PRG_Gauge, it is redanduncy and make sure change the PRG_Gauge as well if change here
    stDREAM_MC_GAUGE := stDREAM_MC_GHC_GAUGE;
    stDREAM_MC_GAUGE.sPath := 'DREAM_MC_GHC_GAUGE';
END_IF

//Select DS interlock gauge
IF NOT DREAM_CAT1_GHC_01.IG.xPRESS_OK THEN
    stDREAM_CAT1_GAUGE := DREAM_ROUGH2_GPI_03.PG;
    stDREAM_CAT1_GAUGE.sPath := 'DREAM_ROUGH2_GPI_03';
ELSE
      stDREAM_CAT1_GAUGE := DREAM_CAT1_GHC_01.IG;
    stDREAM_CAT1_GAUGE.sPath := 'DREAM_CAT1_GHC_01';
END_IF

bCAT1_VRC_01_ExtILK := bCAT1_VRC_01_ExtILK_US AND bCATPumpsRunning;

//DREAM_CAT1_VRC_01(i_xExtILK_OK := bCAT1_VRC_01_ILK, i_xOverrideMode := bSystemOverrideMode);
DREAM_CAT1_VRC_01(i_stUSG := stDREAM_MC_GAUGE,
                  i_stDSG := stDREAM_CAT1_GAUGE,
                  i_xDis_DPIlk := FALSE,
                  i_xEPS_OK := TRUE,
                  i_xPMPS_OK := TRUE,
                  i_xReset := FALSE,
                  i_xExt_OK := bCAT1_VRC_01_ExtILK,
                  i_xOverrideMode := bSystemOverrideMode,
                  io_fbFFHWO := dummy_FFFO,
                  fbArbiter := dummy_fbArbiter1,
                  i_sDevName := 'DREAM-CAT1-VRC-01');

(**Roughing Valves**)
//Interlock evaluation
bROUGH1_VRC_01_ILK := //DREAM_ROUGH1_GPI_01.PG.rPRESS < 5E-3 AND DREAM_ROUGH1_GPI_01.PG.xPRESS_OK AND
                      DREAM_ROUGH1_VFV_01.iq_stVFN.rReqPosition = 0.0 AND
                      DREAM_ROUGH1_VFV_02.iq_stVFN.rReqPosition = 0.0 AND
                      DREAM_ROUGH1_VRC_10.iq_stValve.i_xClsLS; //Interlocked with manifold roughing valve as well

bROUGH2_VRC_01_ILK := //DREAM_ROUGH2_GPI_01.PG.rPRESS < 5E-3 AND DREAM_ROUGH2_GPI_01.PG.xPRESS_OK AND
                      DREAM_ROUGH2_VFV_01.iq_stVFN.rReqPosition = 0.0 AND
                      DREAM_ROUGH2_VFV_02.iq_stVFN.rReqPosition = 0.0;

bROUGH2_VRC_02_ILK := //DREAM_ROUGH2_GPI_01.PG.rPRESS < 5E-3 AND DREAM_ROUGH2_GPI_01.PG.xPRESS_OK AND
                      DREAM_ROUGH2_VFV_01.iq_stVFN.rReqPosition = 0.0 AND
                      DREAM_ROUGH2_VFV_03.iq_stVFN.rReqPosition = 0.0;

bROUGH1_VRC_01_Override := bSystemOverrideMode AND
                           DREAM_ROUGH1_VFV_01.iq_stVFN.rReqPosition = 0.0 AND
                           DREAM_ROUGH1_VFV_02.iq_stVFN.rReqPosition = 0.0;

bROUGH2_VRC_01_Override := bSystemOverrideMode AND
                           DREAM_ROUGH2_VFV_01.iq_stVFN.rReqPosition = 0.0 AND
                           DREAM_ROUGH2_VFV_02.iq_stVFN.rReqPosition = 0.0;

bROUGH2_VRC_02_Override := bSystemOverrideMode AND
                           DREAM_ROUGH2_VFV_01.iq_stVFN.rReqPosition = 0.0 AND
                           DREAM_ROUGH2_VFV_03.iq_stVFN.rReqPosition = 0.0;

DREAM_ROUGH1_VRC_01(i_stUSG := DREAM_ROUGH1_GPI_01.PG,
                    i_stDSG := DREAM_ROUGH1_GPI_02.PG,
                    i_xDis_DPIlk := FALSE,
                    i_xEPS_OK := TRUE,
                    i_xPMPS_OK := TRUE,
                    i_xReset := FALSE,
                    i_xExt_OK := bROUGH1_VRC_01_ILK,
                    i_xOverrideMode := bROUGH1_VRC_01_Override,
                    io_fbFFHWO := dummy_FFFO,
                    fbArbiter := dummy_fbArbiter1,
                    i_sDevName := 'DREAM-ROUGH1-VRC-01');

DREAM_ROUGH2_VRC_01(i_stUSG := DREAM_ROUGH2_GPI_01.PG,
                    i_stDSG := DREAM_ROUGH2_GPI_02.PG,
                    i_xDis_DPIlk := FALSE,
                    i_xEPS_OK := TRUE,
                    i_xPMPS_OK := TRUE,
                    i_xReset := FALSE,
                    i_xExt_OK := bROUGH2_VRC_01_ILK,
                    i_xOverrideMode := bROUGH2_VRC_01_Override,
                    io_fbFFHWO := dummy_FFFO,
                    fbArbiter := dummy_fbArbiter1,
                    i_sDevName := 'DREAM-ROUGH2-VRC-01');

DREAM_ROUGH2_VRC_02(i_stUSG := DREAM_ROUGH2_GPI_01.PG,
                    i_stDSG := DREAM_ROUGH2_GPI_03.PG,
                    i_xDis_DPIlk := FALSE,
                    i_xEPS_OK := TRUE,
                    i_xPMPS_OK := TRUE,
                    i_xReset := FALSE,
                    i_xExt_OK := bROUGH2_VRC_02_ILK,
                    i_xOverrideMode := bROUGH2_VRC_02_Override,
                    io_fbFFHWO := dummy_FFFO,
                    fbArbiter := dummy_fbArbiter1,
                    i_sDevName := 'DREAM-ROUGH2-VRC-02');

//Test valve
DREAM_ROUGH1_VRC_20(i_xExtILK_OK := True, i_xOverrideMode := bSystemOverrideMode);

//Manifold roughing valve
DREAM_ROUGH1_VRC_10(i_xExtILK_OK := DREAM_ROUGH1_VRC_01.iq_stValve.i_xClsLS, i_xOverrideMode := bSystemOverrideMode);

//Flow control valves
DREAM_ROUGH1_VFV_01(i_xExtIlkOK := DREAM_ROUGH1_VRC_01.iq_stValve.i_xClsLS);

DREAM_ROUGH1_VFV_02(i_xExtIlkOK := DREAM_ROUGH1_VRC_01.iq_stValve.i_xClsLS AND DREAM_DP1_VRC_01.iq_stValve.i_xClsLS AND
                                   NOT DREAM_NC_PTM_01.iq_stPTM.i_xAtSpd AND
                                   NOT DREAM_NC_PTM_02.iq_stPTM.i_xAtSpd);

DREAM_ROUGH2_VFV_01(i_xExtIlkOK := DREAM_ROUGH2_VRC_01.iq_stValve.i_xClsLS AND DREAM_ROUGH2_VRC_02.iq_stValve.i_xClsLS);

DREAM_ROUGH2_VFV_02(i_xExtIlkOK := DREAM_ROUGH2_VRC_01.iq_stValve.i_xClsLS AND
                                   NOT DREAM_DP1_PTM_01.iq_stPTM.i_xAtSpd AND
                                   NOT DREAM_DP2_PTM_01.iq_stPTM.i_xAtSpd AND
                                   NOT DREAM_DP3_PTM_01.iq_stPTM.i_xAtSpd AND
                                   NOT DREAM_MC_PTM_01.iq_stPTM.i_xAtSpd AND
                                   NOT DREAM_MC_PTM_02.iq_stPTM.i_xAtSpd AND
                                   NOT DREAM_ROUGH2_PTM_01.iq_stPTM.i_xAtSpd AND
                                   NOT DREAM_ROUGH2_PTM_02.iq_stPTM.i_xAtSpd AND
                                   NOT DREAM_CAT1_PTM_01.iq_stPTM.i_xAtSpd);

DREAM_ROUGH2_VFV_03(i_xExtIlkOK := DREAM_ROUGH2_VRC_02.iq_stValve.i_xClsLS AND DREAM_CAT1_VRC_01.iq_stValve.i_xClsLS AND
                                   NOT DREAM_CAT2_PTM_01.iq_stPtm.i_xAtSpd);

//dual vale for test-08-15-25
DREAM_DP1_VRC_20(i_OPN_OK := TRUE,
                 i_CLS_OK := TRUE,
                 ibCntrlHold := FALSE,
                 i_xOverrideMode :=  bSystemOverrideMode,
                 iq_stValve =>);

END_PROGRAM

// ---- POUs/PRG_TURBO_PUMPS.TcPOU
PROGRAM PRG_TURBO_PUMPS
VAR
    bAllTurboPumpRunning : BOOL;
    tAllTurboPumpDelayTime : TIME := T#30s;
    tAllTurboPumpTOF : TOF;

    bMainTurboPumpRunning : BOOL;
    tMainTurboPumpDelayTime : TIME := T#15m;
    tMainTurboPumpTOF : TOF;
    ftPumpsFailed : F_TRIG;
END_VAR

(**Gas Injection Turbo pumps**)
DREAM_NC_PTM_01(i_xExtIlkOK := DREAM_ROUGH1_GPI_02.PG.rPRESS < DREAM_NC_PTM_01.iq_stPTM.rBackingPressureSP AND DREAM_ROUGH1_GPI_02.PG.xPRESS_OK AND
                               DREAM_ROUGH1_VRC_01.iq_stValve.i_xOpnLS);

DREAM_NC_PTM_02(i_xExtIlkOK := DREAM_ROUGH1_GPI_02.PG.rPRESS < DREAM_NC_PTM_02.iq_stPTM.rBackingPressureSP AND DREAM_ROUGH1_GPI_02.PG.xPRESS_OK AND
                               DREAM_ROUGH1_VRC_01.iq_stValve.i_xOpnLS);

(**Differential pumping stations Turbo pumps**)
DREAM_DP1_PTM_01(i_xExtIlkOK := DREAM_ROUGH2_GPI_02.PG.rPRESS < DREAM_DP1_PTM_01.iq_stPTM.rBackingPressureSP AND DREAM_ROUGH2_GPI_02.PG.xPRESS_OK AND
                                DREAM_ROUGH2_VRC_01.iq_stValve.i_xOpnLS);

DREAM_DP2_PTM_01(i_xExtIlkOK := DREAM_ROUGH2_GPI_02.PG.rPRESS < DREAM_DP2_PTM_01.iq_stPTM.rBackingPressureSP AND DREAM_ROUGH2_GPI_02.PG.xPRESS_OK AND
                                DREAM_ROUGH2_VRC_01.iq_stValve.i_xOpnLS);

DREAM_DP3_PTM_01(i_xExtIlkOK := DREAM_ROUGH2_GPI_02.PG.rPRESS < DREAM_DP3_PTM_01.iq_stPTM.rBackingPressureSP AND DREAM_ROUGH2_GPI_02.PG.xPRESS_OK AND
                                DREAM_ROUGH2_VRC_01.iq_stValve.i_xOpnLS);

(**Main Chamber Turbo pumps**)
DREAM_MC_PTM_01(i_xExtIlkOK := DREAM_ROUGH2_GPI_02.PG.rPRESS < DREAM_MC_PTM_01.iq_stPTM.rBackingPressureSP AND DREAM_ROUGH2_GPI_02.PG.xPRESS_OK AND
                               DREAM_ROUGH2_VRC_01.iq_stValve.i_xOpnLS);

DREAM_MC_PTM_02(i_xExtIlkOK := DREAM_ROUGH2_GPI_02.PG.rPRESS < DREAM_MC_PTM_02.iq_stPTM.rBackingPressureSP AND DREAM_ROUGH2_GPI_02.PG.xPRESS_OK AND
                               DREAM_ROUGH2_VRC_01.iq_stValve.i_xOpnLS);

(**Catcher Turbo pumps**)
//Special interlock due to manual valve between turbo pump and ROUGH2_GPI2
DREAM_CAT1_PTM_01(i_xExtIlkOK := DREAM_ROUGH2_GPI_02.PG.rPRESS < DREAM_CAT1_PTM_01.iq_stPTM.rBackingPressureSP AND DREAM_ROUGH2_GPI_02.PG.xPRESS_OK AND
                                 DREAM_ROUGH2_GPI_03.PG.rPRESS < DREAM_CAT1_PTM_01.iq_stPTM.rBackingPressureSP AND DREAM_ROUGH2_GPI_03.PG.xPRESS_OK AND
                                 DREAM_ROUGH2_VRC_01.i_xOpnLS);


DREAM_CAT2_PTM_01(i_xExtIlkOK := DREAM_ROUGH2_GPI_03.PG.rPRESS < DREAM_CAT2_PTM_01.iq_stPTM.rBackingPressureSP AND DREAM_ROUGH2_GPI_03.PG.xPRESS_OK AND
                                 DREAM_ROUGH2_VRC_02.iq_stValve.i_xOpnLS);

(**ROUGHING SECTION TURBO BOOSTER PUMPS**)
DREAM_ROUGH2_PTM_01(i_xExtIlkOK := DREAM_ROUGH2_GPI_02.PG.rPRESS < DREAM_ROUGH2_PTM_01.iq_stPTM.rBackingPressureSP AND DREAM_ROUGH2_GPI_02.PG.xPRESS_OK AND
                                   DREAM_ROUGH2_VRC_01.iq_stValve.i_xOpnLS);

DREAM_ROUGH2_PTM_02(i_xExtIlkOK := DREAM_ROUGH2_GPI_02.PG.rPRESS < DREAM_ROUGH2_PTM_02.iq_stPTM.rBackingPressureSP AND DREAM_ROUGH2_GPI_02.PG.xPRESS_OK AND
                                   DREAM_ROUGH2_VRC_01.iq_stValve.i_xOpnLS);


bAllTurboPumpRunning := DREAM_NC_PTM_01.iq_stPTM.eState = E_PumpState.pumpRUNNING AND
                        DREAM_NC_PTM_02.iq_stPTM.eState = E_PumpState.pumpRUNNING AND
                        DREAM_DP1_PTM_01.iq_stPTM.eState = E_PumpState.pumpRUNNING AND
                        DREAM_DP2_PTM_01.iq_stPTM.eState = E_PumpState.pumpRUNNING AND
                        DREAM_DP3_PTM_01.iq_stPTM.eState = E_PumpState.pumpRUNNING AND
                        DREAM_MC_PTM_01.iq_stPTM.eState = E_PumpState.pumpRUNNING AND
                        DREAM_MC_PTM_02.iq_stPTM.eState = E_PumpState.pumpRUNNING AND
                        DREAM_CAT1_PTM_01.iq_stPTM.eState = E_PumpState.pumpRUNNING AND
                        DREAM_CAT2_PTM_01.iq_stPTM.eState = E_PumpState.pumpRUNNING AND
                        DREAM_ROUGH2_PTM_01.iq_stPTM.eState = E_PumpState.pumpRUNNING AND
                        DREAM_ROUGH2_PTM_02.iq_stPTM.eState = E_PumpState.pumpRUNNING;

tAllTurboPumpTOF(IN := bAllTurboPumpRunning, PT := tAllTurboPumpDelayTime);
bDREAM_TURBOS_ALL_AtSpd := tAllTurboPumpTOF.Q;

bMCPumpsRunning := DREAM_DP1_PTM_01.iq_stPTM.eState = E_PumpState.pumpRUNNING AND
                   DREAM_DP2_PTM_01.iq_stPTM.eState = E_PumpState.pumpRUNNING AND
                   DREAM_DP3_PTM_01.iq_stPTM.eState = E_PumpState.pumpRUNNING AND
                   DREAM_MC_PTM_01.iq_stPTM.eState = E_PumpState.pumpRUNNING AND
                   DREAM_MC_PTM_02.iq_stPTM.eState = E_PumpState.pumpRUNNING AND
                   DREAM_ROUGH2_PTM_01.iq_stPTM.eState = E_PumpState.pumpRUNNING AND
                   DREAM_ROUGH2_PTM_02.iq_stPTM.eState = E_PumpState.pumpRUNNING;

bCATPumpsRunning := DREAM_CAT1_PTM_01.iq_stPTM.eState = E_PumpState.pumpRUNNING AND
                    DREAM_CAT2_PTM_01.iq_stPTM.eState = E_PumpState.pumpRUNNING;

(*********SERIAL COMMUNICATION**********)

(*Pfeiffer pumps at Gas Injection*)
//DREAM_NC_PTM_01
(*Assign adresses to the pfeiffer controllers connected to this serial terminal*)
stPfeiffer_CTRL_DREAM_NC_PTM_01[1].iSerialAddress:= 1;
stPfeiffer_CTRL_DREAM_NC_PTM_01[1].xEnableComm:= TRUE;
(*Instanitate the Function block for serial communication with Pfeiffer*)
fbPfeifferCom_DREAM_NC_PTM_01(astPfeifferControl:= stPfeiffer_CTRL_DREAM_NC_PTM_01,
                              astPfeifferStatus:= stPfeiffer_RBK_DREAM_NC_PTM_01,
                              SerialRXBuffer:= SerialRXBuffer_DREAM_NC_PTM_01,
                              SerialTXBuffer:= SerialTXBuffer_DREAM_NC_PTM_01);
(*Copy Status Pv's into the PTM structure*)
DREAM_NC_PTM_01.M_Serial_IO(st_Pfeiffer_RBK:= stPfeiffer_RBK_DREAM_NC_PTM_01[1],
                            st_Pfeiffer_CTRL:= stPfeiffer_CTRL_DREAM_NC_PTM_01[1]);

//DREAM_NC_PTM_02
stPfeiffer_CTRL_DREAM_NC_PTM_02[1].iSerialAddress:= 1;
stPfeiffer_CTRL_DREAM_NC_PTM_02[1].xEnableComm:= TRUE;
fbPfeifferCom_DREAM_NC_PTM_02(astPfeifferControl:= stPfeiffer_CTRL_DREAM_NC_PTM_02,
                              astPfeifferStatus:= stPfeiffer_RBK_DREAM_NC_PTM_02,
                              SerialRXBuffer:= SerialRXBuffer_DREAM_NC_PTM_02,
                              SerialTXBuffer:= SerialTXBuffer_DREAM_NC_PTM_02);

DREAM_NC_PTM_02.M_Serial_IO(st_Pfeiffer_RBK:= stPfeiffer_RBK_DREAM_NC_PTM_02[1],
                            st_Pfeiffer_CTRL:= stPfeiffer_CTRL_DREAM_NC_PTM_02[1]);

//DREAM_DP1_PTM_01
stPfeiffer_CTRL_DREAM_DP1_PTM_01[1].iSerialAddress:= 1;
stPfeiffer_CTRL_DREAM_DP1_PTM_01[1].xEnableComm:= TRUE;
fbPfeifferCom_DREAM_DP1_PTM_01(astPfeifferControl:= stPfeiffer_CTRL_DREAM_DP1_PTM_01,
                               astPfeifferStatus:= stPfeiffer_RBK_DREAM_DP1_PTM_01,
                               SerialRXBuffer:= SerialRXBuffer_DREAM_DP1_PTM_01,
                               SerialTXBuffer:= SerialTXBuffer_DREAM_DP1_PTM_01);

DREAM_DP1_PTM_01.M_Serial_IO(st_Pfeiffer_RBK:= stPfeiffer_RBK_DREAM_DP1_PTM_01[1],
                             st_Pfeiffer_CTRL:= stPfeiffer_CTRL_DREAM_DP1_PTM_01[1]);


(*Leybold pumps at Gas Injection*)
//DREAM_DP2_PTM_01
(*Instanitate the Function block for serial communication with TD20 controller*)
fbTD20Com_DREAM_DP2_PTM_01(SerialRXBuffer:= SerialRXBuffer_DREAM_DP2_PTM_01,
                           SerialTXBuffer:= SerialTXBuffer_DREAM_DP2_PTM_01,
                           astTD20Status=> stTD20_RBK_DREAM_DP2_PTM_01);
(*Copy Status Pv's into the PTM structure*)
DREAM_DP2_PTM_01.M_Serial_IO(i_st_TD20_RBK:= stTD20_RBK_DREAM_DP2_PTM_01);

//DREAM_DP3_PTM_01
fbTD20Com_DREAM_DP3_PTM_01(SerialRXBuffer:= SerialRXBuffer_DREAM_DP3_PTM_01,
                           SerialTXBuffer:= SerialTXBuffer_DREAM_DP3_PTM_01,
                           astTD20Status=> stTD20_RBK_DREAM_DP3_PTM_01);

DREAM_DP3_PTM_01.M_Serial_IO(i_st_TD20_RBK:= stTD20_RBK_DREAM_DP3_PTM_01);

(*Leybold pumps at Main Chamber*)
//DREAM_MC_PTM_01
fbTD20Com_DREAM_MC_PTM_01(SerialRXBuffer:= SerialRXBuffer_DREAM_MC_PTM_01,
                           SerialTXBuffer:= SerialTXBuffer_DREAM_MC_PTM_01,
                           astTD20Status=> stTD20_RBK_DREAM_MC_PTM_01);

DREAM_MC_PTM_01.M_Serial_IO(stTD20_RBK_DREAM_MC_PTM_01);

//DREAM_MC_PTM_02
fbTD20Com_DREAM_MC_PTM_02(SerialRXBuffer:= SerialRXBuffer_DREAM_MC_PTM_02,
                           SerialTXBuffer:= SerialTXBuffer_DREAM_MC_PTM_02,
                           astTD20Status=> stTD20_RBK_DREAM_MC_PTM_02);

DREAM_MC_PTM_02.M_Serial_IO(stTD20_RBK_DREAM_MC_PTM_02);

(*Leybold pumps at Catcher*)
//DREAM_CAT1_PTM_01 (TD400)
fbTD400SerialIO_DREAM_CAT1_PTM_01(iq_stPTM := DREAM_CAT1_PTM_01.iq_stPtm,
                                  iq_stTD400Control := stTD400_CTRL_DREAM_CAT1_PTM_01,
                                  iq_stTD400Status := stTD400_RBK_DREAM_CAT1_PTM_01);

fbTD400Com_DREAM_CAT1_PTM_01(SerialRXBuffer := SerialRXBuffer_DREAM_CAT1_PTM_01,
                             SerialTXBuffer := SerialTXBuffer_DREAM_CAT1_PTM_01,
                             stTD400Control := stTD400_CTRL_DREAM_CAT1_PTM_01,
                             stTD400Status => stTD400_RBK_DREAM_CAT1_PTM_01);

//DREAM_CAT1_PTM_01.M_Serial_IO(stTD400_RBK_DREAM_CAT1_PTM_01);

//DREAM_CAT2_PTM_01 (TD400)
fbTD400SerialIO_DREAM_CAT2_PTM_01(iq_stPTM := DREAM_CAT2_PTM_01.iq_stPtm,
                                  iq_stTD400Control := stTD400_CTRL_DREAM_CAT2_PTM_01,
                                  iq_stTD400Status := stTD400_RBK_DREAM_CAT2_PTM_01);

fbTD400Com_DREAM_CAT2_PTM_01(SerialRXBuffer := SerialRXBuffer_DREAM_CAT2_PTM_01,
                             SerialTXBuffer := SerialTXBuffer_DREAM_CAT2_PTM_01,
                             stTD400Control := stTD400_CTRL_DREAM_CAT2_PTM_01,
                             stTD400Status => stTD400_RBK_DREAM_CAT2_PTM_01);

//DREAM_CAT2_PTM_01.M_Serial_IO(stTD400_RBK_DREAM_CAT2_PTM_01);

(*Leybold pump-roughing section-booster pump*)
//DREAM_ROUGH2_PTM_01 (TD400)
fbTD400SerialIO_DREAM_ROUGH2_PTM_01(iq_stPTM := DREAM_ROUGH2_PTM_01.iq_stPtm,
                                    iq_stTD400Control := stTD400_CTRL_DREAM_ROUGH2_PTM_01,
                                    iq_stTD400Status := stTD400_RBK_DREAM_ROUGH2_PTM_01);

fbTD400Com_DREAM_ROUGH2_PTM_01(SerialRXBuffer := SerialRXBuffer_DREAM_ROUGH2_PTM_01,
                               SerialTXBuffer := SerialTXBuffer_DREAM_ROUGH2_PTM_01,
                               stTD400Control := stTD400_CTRL_DREAM_ROUGH2_PTM_01,
                               stTD400Status => stTD400_RBK_DREAM_ROUGH2_PTM_01);

//DREAM_ROUGH2_PTM_01.M_Serial_IO(stTD400_RBK_DREAM_ROUGH2_PTM_01);

//DREAM_ROUGH2_PTM_01 (TD400)
fbTD400SerialIO_DREAM_ROUGH2_PTM_02(iq_stPTM := DREAM_ROUGH2_PTM_02.iq_stPtm,
                                    iq_stTD400Control := stTD400_CTRL_DREAM_ROUGH2_PTM_02,
                                    iq_stTD400Status := stTD400_RBK_DREAM_ROUGH2_PTM_02);

fbTD400Com_DREAM_ROUGH2_PTM_02(SerialRXBuffer := SerialRXBuffer_DREAM_ROUGH2_PTM_02,
                               SerialTXBuffer := SerialTXBuffer_DREAM_ROUGH2_PTM_02,
                               stTD400Control := stTD400_CTRL_DREAM_ROUGH2_PTM_02,
                               stTD400Status => stTD400_RBK_DREAM_ROUGH2_PTM_02);

//DREAM_ROUGH2_PTM_02.M_Serial_IO(stTD400_RBK_DREAM_ROUGH2_PTM_02);

END_PROGRAM

// ---- POUs/PRG_HV_ILK.TcPOU
PROGRAM PRG_HV_ILK
VAR

END_VAR

(*High Voltage Saftey Loop*)
IF GVL_VAC_GAUGES.stDREAM_MC_GHC_GAUGE.xPRESS_OK THEN
  //  fHighVoltageMaxPressure := 1e-05;
    GVL_PLC_Interface.bHVSafteyLoopEnable := GVL_VAC_GAUGES.stDREAM_MC_GHC_GAUGE.rPRESS <= fHighVoltageMaxPressure;
ELSIF DREAM_MC_GPI_01.PG.xPRESS_OK AND bMCPumpsRunning THEN
 //   fHighVoltageMaxPressure := 5e-04;
    GVL_PLC_Interface.bHVSafteyLoopEnable := DREAM_MC_GPI_01.PG.rPRESS <= rHV_GPI_SP;
ELSE
    GVL_PLC_Interface.bHVSafteyLoopEnable := FALSE;
END_IF

END_PROGRAM

// ---- POUs/PRG_COIL_PS_ILK.TcPOU
PROGRAM PRG_COIL_PS_ILK
VAR
END_VAR

(*Interlock logic for Coil PS based on reading from Flow meter*)
fbCoilFlowMeter();
fCoilCoolantFlowMeterRBV := fbCoilFlowMeter.fReal;

//evaluate flow meter readback to Interlock interlock Coil PS
bCoilPS_ILK := fbCoilFlowMeter.fReal > 3.0; //If flow meter reading is above XX is ok to turn ON output of the Coil PS. Units are lpm

//fbDreamCoilFlowMeter();
//bCoilPS_ILK := fbDreamCoilFlowMeter.fbFlowMeter.fReal > 3; //If flow meter reading is above XX is ok to turn ON output of the Coil PS. Units are lpm

(*DREAM Coil PS Current Monitoring*)
fbCoilCurrentMonitoring();
fCoilCurrentRBV := fbCoilCurrentMonitoring.fReal;

END_PROGRAM

// ---- POUs/PRG_TC.TcPOU
PROGRAM PRG_TC
VAR
END_VAR

//Measure Thercmocouples
TC_01();
TC_02();
TC_03();
TC_04();
TC_05();
TC_06();
TC_07();
TC_08();

END_PROGRAM

// ---- POUs/PRG_AUTOMATION.TcPOU
PROGRAM PRG_AUTOMATION
VAR
    eCurrOp : E_Op; // Currently running operation
    fbVentMcCat : FB_VentMcCat;
    fbAtVacuum : FB_AtVacuum;
END_VAR

(* Run operations, but don't start any new operations if another operation is still running or error is present *)
// Reset error
IF GVL_Automation.i_bResetError THEN
    GVL_Automation.q_bError := FALSE;
    GVL_Automation.i_bResetError := FALSE;
END_IF

// Only start new operations if the system is NOT busy with another operation and transtion to new state is valid and no error present
IF NOT GVL_Automation.q_bBusy AND NOT GVL_Automation.q_bError THEN
    IF F_IsValidStateTransition(eCurrOp, GVL_Automation.iq_eOperation) THEN
        eCurrOp := GVL_Automation.iq_eOperation;
    ELSE
        GVL_Automation.q_sMessage := 'Invalid state transition';
        //GVL_Automation.q_bError := TRUE;
    END_IF
END_IF

// Execute selected operation
CASE eCurrOp OF
E_Op.INIT: // State Machine INIT // do nothing for now, can be used in the future if needed
    eCurrOp := E_Op.STANDBY;
    GVL_Automation.q_sMessage := 'Initialization completed';

E_Op.STANDBY: // Monitoring IF full system under vacuum
    GVL_Automation.q_bBusy := FALSE;
    (*IF F_AllPumpsRunning() AND F_PressAtVacSP() AND NOT GVL_Automation.q_bError THEN // clear the error before start monitoring again
        eCurrOp := E_Op.AT_VACUUM;
        GVL_Automation.q_bBusy := TRUE; // Extend for one cycle so the state doesn't get overrired
        GVL_Automation.q_sMessage := 'MC At Vacuum';
    END_IF*)

E_Op.PUMP_ALL: // Full system pump down
    GVL_Automation.q_bBusy := FALSE; //do nothing for now, will be implemented later. When pumping down procedure ends go to xxxxxx state

E_Op.PUMP_NC: // Only Nozzle chamber pump down
    GVL_Automation.q_bBusy := FALSE; // do nothing for now, will be implemented later. When pumping down procedure of NC only ends go back to Standby state

E_Op.AT_VACUUM: // Monitor if system is At Vacuum (pumps running and pressure below SP), if vaccum event occurs vent full system
    fbAtVacuum(
        i_bExecute := TRUE,
        i_bCancel := GVL_Automation.i_bCancel,
        iq_sMessageBuffer := GVL_Automation.q_sMessage,
        q_bBusy => GVL_Automation.q_bBusy,
        q_bError => GVL_Automation.q_bError
    );
    IF GVL_Automation.q_bError THEN // Vent MC and CAT IF Vacuum fault on main chamber detected
        eCurrOp := E_Op.VENT_MC_CAT;
        GVL_Automation.q_bBusy := TRUE; // Extend for one cycle so the eCurrOp doesn't get overried
    END_IF

E_Op.VENT_ALL: // Vent full system
    GVL_Automation.q_bBusy := FALSE; // do nothing for now, will be implemented later

E_Op.VENT_NC: // Vent nozzle chamber only
    GVL_Automation.q_bBusy := FALSE; // do nothing for now, will be implemented later

E_Op.VENT_MC_CAT: // Vent Main Chamber + Catcher
    (*fbVentMcCat(
        i_bExecute := TRUE,
        i_bCancel := GVL_Automation.i_bCancel,
        iq_sMessageBuffer := GVL_Automation.q_sMessage,
        q_bBusy => GVL_Automation.q_bBusy,
        q_bError => GVL_Automation.q_bError
    );*)
    GVL_Automation.q_bBusy := FALSE; //temporary before enabling code above

E_Op.VENT_CAT: // Vent catcher only
    GVL_Automation.q_bBusy := FALSE; // do nothing for now, will be implemented later

ELSE // Selected unimplemented operation
    GVL_Automation.q_sMessage := 'Unimplemented operation';
    GVL_Automation.q_bBusy := FALSE;
    GVL_Automation.q_bError := TRUE;
END_CASE

// If all operation have finished then go back to standby
IF NOT GVL_Automation.q_bBusy THEN
    eCurrOp := E_Op.STANDBY;
END_IF

// Set output operation to whatever is ACTAULLY currently running
GVL_Automation.iq_eOperation := eCurrOp;
GVL_Automation.i_bCancel := FALSE; // Reset cancel flag

END_PROGRAM

// ---- POUs/Automation/FB_VentMcCat.TcPOU
FUNCTION_BLOCK FB_VentMcCat EXTENDS FB_Operation
VAR_INPUT
END_VAR
VAR_OUTPUT
END_VAR
VAR
    fRough2VFV2Position : REAL;
    fRough2VFV3Position : REAL;
END_VAR
VAR CONSTANT
    VFV_MAX_POSITION : INT := 100;
END_VAR

SUPER^(iq_sMessageBuffer := iq_sMessageBuffer);

// Think which steps should not be permitted to cancel, figure out during testing
CASE eStep OF
E_OpStep.IDLE: // Do nothing

E_OpStep.START: // Close beamline window valves //Defer cancel if this procedure should not be cancelled from user!
    // Close window beamline valves
    GVL_PLC_Interface.bCLOSE_TMO_MR5K4_VWC := TRUE;
    GVL_PLC_Interface.bCLOSE_TMO_TM2K4_VWC := TRUE;
    M_SetMessage('Closing TMO window valves');
    M_RunTimeoutTimer(VALVE_TIMEOUT);

    IF (GVL_PLC_Interface.bTMO_MR5K4_VWC_CLOSED_LS AND GVL_PLC_Interface.bTMO_TM2K4_VWC_CLOSED_LS) THEN
        M_SetMessage('Window valves closed');
        M_ResetTimeoutTimer();
        eStep := E_OpStep.VMCAS_CLOSE_ISOLATION_VALVES;
    ELSIF M_TimeoutExpired() THEN
        M_SetMessage('Closing window valve - timeout');
        M_ResetTimeoutTimer();
        eStep := E_OpStep.VMCAS_CLOSE_ISOLATION_VALVES;
    END_IF

E_OpStep.VMCAS_CLOSE_ISOLATION_VALVES: // Close isolation valves (DP1:VRC:01, CAT1:VRC:01), Bypas valve DP1:VRC:01 shall open
    DREAM_DP1_VRC_01.M_Set_OPN_SW(FALSE);
    DREAM_CAT1_VRC_01.M_Set_OPN_SW(FALSE);
    M_SetMessage('Close Isolation valves');
    M_RunTimeoutTimer(VALVE_TIMEOUT);

    IF DREAM_DP1_VRC_01.iq_stValve.i_xClsLS AND DREAM_CAT1_VRC_01.iq_stValve.i_xClsLS AND DREAM_DP1_VRC_02.iq_stValve.i_xOpnLS THEN
        M_SetMessage('Isolation valves closed, bypass open');
        M_ResetTimeoutTimer();
        eStep := E_OpStep.VMCAS_STOP_TURBO_PUMPS;
    ELSIF M_TimeoutExpired() THEN
        M_FatalError('Moving isolation,bypass valves-timeout'); // Raise the error, don't move forward with stopping pumps etc.
    END_IF

E_OpStep.VMCAS_STOP_TURBO_PUMPS: // Stop MC and CAT Turbo pumps
    DREAM_DP1_PTM_01.M_Run(FALSE);
    DREAM_DP2_PTM_01.M_Run(FALSE);
    DREAM_DP3_PTM_01.M_Run(FALSE);
    DREAM_MC_PTM_01.M_Run(FALSE);
    DREAM_MC_PTM_02.M_Run(FALSE);
    DREAM_CAT1_PTM_01.M_Run(FALSE);
    DREAM_CAT2_PTM_01.M_Run(FALSE);
    DREAM_ROUGH2_PTM_01.M_Run(FALSE);
    DREAM_ROUGH2_PTM_02.M_Run(FALSE);

    M_SetMessage('Stopping MC and CAT turbos');
    eStep := E_OpStep.VMCAS_CLOSE_ROUGH_VALVES;

E_OpStep.VMCAS_CLOSE_ROUGH_VALVES: // Close roughing valves
    DREAM_ROUGH2_VRC_01.M_Set_OPN_SW(FALSE);
    DREAM_ROUGH2_VRC_02.M_Set_OPN_SW(FALSE);
    M_SetMessage('Close Roughing valves');
    M_RunTimeoutTimer(VALVE_TIMEOUT);

    IF DREAM_ROUGH2_VRC_01.iq_stValve.i_xClsLS AND DREAM_ROUGH2_VRC_02.iq_stValve.i_xClsLS THEN
        M_SetMessage('Roughing valves closed');
        M_ResetTimeoutTimer();
        eStep := E_OpStep.VMCAS_STOP_GAUGES;
    ELSIF M_TimeoutExpired() THEN
        M_FatalError('Moving roughing valves-timeout'); // Raise the error, don't move forward with stopping gauges etc.
    END_IF

E_OpStep.VMCAS_STOP_GAUGES: // Turn off gauges // I'm thinking to move this state to before closing rough valves becasue in previos state if error is raised gauges will remain ON while pumps already stopped
    DREAM_DP1_GHC_01.M_HVE(FALSE);
    DREAM_DP2_GHC_01.M_HVE(FALSE);
    DREAM_DP3_GHC_01.M_HVE(FALSE);
    DREAM_MC_GHC.M_HVECh1(FALSE);
    DREAM_MC_GHC.M_HVECh2(FALSE);
    DREAM_CAT1_GHC_01.M_HVE(FALSE);
    DREAM_CAT2_GHC_01.M_HVE(FALSE);

    M_SetMessage('Turning OFF MC and CAT Gauges');
    eStep := E_OpStep.VMCAS_WAIT_FOR_TURBO_PUMPS_SPIN_DOWN;

E_OpStep.VMCAS_WAIT_FOR_TURBO_PUMPS_SPIN_DOWN: // Turbos need to spin down to below 100 Hz before start venting procedure
    M_RunTimeoutTimer(TURBOS_SPINDOWN_TIMEOUT); // Timeout is 60 min for now. With testing verify that 30 min is long enough to spin down or increase if needed.
    M_SetMessage('Waiting for pumps to spindown');

    //How should we verify if serial communication work?
    IF DREAM_DP1_PTM_01.iq_stPTM.i_diCurSpd < 100 AND NOT fbSerialLineControl_DREAM_DP1_PTM_01.Error
        AND DREAM_DP2_PTM_01.iq_stPTM.i_diCurSpd < 100 AND NOT fbSerialLineControl_DREAM_DP2_PTM_01.Error
        AND DREAM_DP3_PTM_01.iq_stPTM.i_diCurSpd < 100 AND NOT fbSerialLineControl_DREAM_DP3_PTM_01.Error
        AND DREAM_MC_PTM_01.iq_stPTM.i_diCurSpd < 100 AND NOT fbSerialLineControl_DREAM_MC_PTM_01.Error
        AND DREAM_MC_PTM_02.iq_stPTM.i_diCurSpd < 100 AND NOT fbSerialLineControl_DREAM_MC_PTM_02.Error
        AND DREAM_CAT1_PTM_01.iq_stPTM.i_diCurSpd < 100 AND NOT fbSerialLineControl_DREAM_CAT1_PTM_01.Error
        AND DREAM_CAT2_PTM_01.iq_stPTM.i_diCurSpd < 100 AND NOT fbSerialLineControl_DREAM_CAT2_PTM_01.Error
        AND DREAM_ROUGH2_PTM_01.iq_stPTM.i_diCurSpd < 100 AND NOT fbSerialLineControl_DREAM_ROUGH2_PTM_01.Error
        AND DREAM_ROUGH2_PTM_02.iq_stPTM.i_diCurSpd < 100 AND NOT fbSerialLineControl_DREAM_ROUGH2_PTM_02.Error
    THEN
        M_SetMessage('Pumps below 100 Hz, start venting');
        M_ResetTimeoutTimer();
        eStep := E_OpStep.VMCAS_VENTING;
    ELSIF M_TimeoutExpired()
        AND NOT DREAM_DP1_PTM_01.iq_stPTM.i_xAtSpd
        AND NOT DREAM_DP2_PTM_01.iq_stPTM.i_xAtSpd
        AND NOT DREAM_DP3_PTM_01.iq_stPTM.i_xAtSpd
        AND NOT DREAM_MC_PTM_01.iq_stPTM.i_xAtSpd
        AND NOT DREAM_MC_PTM_02.iq_stPTM.i_xAtSpd
        AND NOT DREAM_CAT1_PTM_01.iq_stPTM.i_xAtSpd
        AND NOT DREAM_CAT2_PTM_01.iq_stPTM.i_xAtSpd
        AND NOT DREAM_ROUGH2_PTM_01.iq_stPTM.i_xAtSpd
        AND NOT DREAM_ROUGH2_PTM_02.iq_stPTM.i_xAtSpd
    THEN (*if serial communication doesn't work and not at speed*)
        M_SetMessage('Pumps spindown-timeout, start venting');
        M_ResetTimeoutTimer();
        eStep := E_OpStep.VMCAS_VENTING;
    ELSE
        M_FatalError('Turbo pumps failed to spin down'); //should I add that state machine goes to error if the pumps didn't start spinning down?
    END_IF

    // Reset vent valve postions
    fRough2VFV2Position := GVL_Constants.ROUGH2_VFV_02_INITIAL_POSITION;
    fRough2VFV3Position := GVL_Constants.ROUGH2_VFV_03_INITIAL_POSITION;

